C07304=1217.053,344.629,-72.947,-176.067,7.468,148.274
C07305=1217.056,344.381,-72.915,-176.068,7.465,148.273
C07306=1217.060,344.133,-72.884,-176.071,7.462,148.273
C07307=1217.065,343.886,-72.851,-176.073,7.460,148.273
C07308=1217.069,343.638,-72.820,-176.074,7.457,148.273
C07309=1217.073,343.389,-72.787,-176.077,7.454,148.273
C07310=1217.078,343.142,-72.756,-176.078,7.451,148.273
C07311=1217.081,342.894,-72.724,-176.080,7.448,148.272
C07312=1217.086,342.646,-72.691,-176.082,7.445,148.272
C07313=1217.090,342.398,-72.660,-176.084,7.442,148.272
C07314=1217.094,342.150,-72.628,-176.086,7.440,148.272
C07315=1217.098,341.902,-72.596,-176.089,7.436,148.272
C07316=1217.102,341.655,-72.564,-176.090,7.434,148.272
C07317=1217.108,341.376,-72.529,-176.092,7.431,148.271
C07318=1217.112,341.099,-72.493,-176.095,7.427,148.271
C07319=1217.117,340.821,-72.457,-176.097,7.424,148.271
C07320=1217.122,340.543,-72.421,-176.099,7.422,148.271
C07321=1217.126,340.294,-72.390,-176.101,7.418,148.271
C07322=1217.130,340.046,-72.358,-176.103,7.416,148.271
C07323=1217.134,339.799,-72.326,-176.105,7.413,148.271
C07324=1217.138,339.551,-72.294,-176.107,7.410,148.270
C07325=1217.142,339.303,-72.263,-176.109,7.407,148.270
C07326=1217.147,339.055,-72.230,-176.111,7.404,148.270
C07327=1217.151,338.806,-72.199,-176.114,7.401,148.270
C07328=1217.155,338.559,-72.168,-176.115,7.399,148.270
C07329=1217.159,338.311,-72.136,-176.117,7.396,148.270
C07330=1217.164,338.063,-72.104,-176.119,7.393,148.269
C07331=1217.168,337.815,-72.072,-176.121,7.391,148.269
C07332=1217.172,337.567,-72.041,-176.123,7.387,148.269
C07333=1217.176,337.319,-72.010,-176.125,7.385,148.269
C07334=1217.180,337.071,-71.978,-176.128,7.382,148.269
C07335=1217.185,336.824,-71.946,-176.129,7.379,148.269
C07336=1217.189,336.575,-71.914,-176.131,7.376,148.269
C07337=1217.193,336.328,-71.883,-176.134,7.374,148.269
C07338=1217.197,336.080,-71.851,-176.136,7.370,148.268
C07339=1217.201,335.831,-71.820,-176.137,7.368,148.268
C07340=1217.205,335.584,-71.789,-176.140,7.366,148.268
C07341=1217.209,335.336,-71.757,-176.142,7.362,148.268
C07342=1217.214,335.087,-71.725,-176.143,7.360,148.268
C07343=1217.218,334.839,-71.693,-176.146,7.357,148.268
C07344=1217.222,334.591,-71.663,-176.148,7.354,148.268
C07345=1217.226,334.343,-71.631,-176.150,7.351,148.267
C07346=1217.230,334.096,-71.599,-176.152,7.349,148.268
C07347=1217.234,333.847,-71.568,-176.154,7.345,148.267
C07348=1217.239,333.600,-71.537,-176.156,7.343,148.267
C07349=1217.243,333.351,-71.506,-176.158,7.340,148.267
C07350=1217.247,333.104,-71.474,-176.160,7.337,148.267
C07351=1217.252,332.855,-71.442,-176.163,7.334,148.267
C07352=1217.256,332.608,-71.411,-176.164,7.332,148.267
C07353=1217.260,332.360,-71.379,-176.167,7.329,148.267
C07354=1217.264,332.112,-71.348,-176.169,7.326,148.267
C07355=1217.268,331.864,-71.317,-176.171,7.324,148.267
C07356=1217.273,331.616,-71.286,-176.173,7.320,148.266
C07357=1217.277,331.367,-71.255,-176.175,7.318,148.266
C07358=1217.281,331.120,-71.223,-176.177,7.315,148.266
C07359=1217.286,330.872,-71.192,-176.179,7.312,148.266
C07360=1217.289,330.624,-71.161,-176.182,7.309,148.266
C07361=1217.294,330.376,-71.130,-176.183,7.307,148.266
C07362=1217.298,330.128,-71.098,-176.186,7.304,148.266
C07363=1217.302,329.880,-71.067,-176.188,7.301,148.266
C07364=1217.306,329.631,-71.036,-176.190,7.298,148.266
C07365=1217.311,329.384,-71.005,-176.192,7.296,148.266
C07366=1217.315,329.136,-70.974,-176.195,7.293,148.266
C07367=1217.319,328.888,-70.942,-176.196,7.290,148.265
C07368=1217.323,328.640,-70.911,-176.198,7.288,148.265
C07369=1217.328,328.391,-70.880,-176.201,7.284,148.265
C07370=1217.332,328.144,-70.849,-176.203,7.282,148.265
C07371=1217.336,327.895,-70.817,-176.205,7.279,148.265
C07372=1217.340,327.647,-70.787,-176.207,7.277,148.265
C07373=1217.344,327.400,-70.756,-176.210,7.274,148.265
C07374=1217.348,327.151,-70.725,-176.211,7.271,148.265
C07375=1217.353,326.904,-70.694,-176.214,7.268,148.265
C07376=1217.357,326.656,-70.663,-176.216,7.266,148.265
C07377=1217.361,326.407,-70.632,-176.218,7.262,148.265
C07378=1217.366,326.160,-70.601,-176.220,7.260,148.265
C07379=1217.370,325.911,-70.569,-176.222,7.257,148.264
C07380=1217.373,325.663,-70.539,-176.225,7.255,148.265
C07381=1217.378,325.415,-70.508,-176.227,7.251,148.264
C07382=1217.382,325.167,-70.477,-176.229,7.249,148.264
C07383=1217.386,324.919,-70.446,-176.232,7.246,148.264
C07384=1217.391,324.671,-70.415,-176.233,7.244,148.264
C07385=1217.395,324.423,-70.384,-176.235,7.241,148.264
C07386=1217.399,324.175,-70.354,-176.238,7.238,148.264
C07387=1217.403,323.927,-70.323,-176.240,7.236,148.264
C07388=1217.408,323.678,-70.292,-176.242,7.233,148.264
C07389=1217.412,323.430,-70.261,-176.244,7.230,148.264
C07390=1217.416,323.183,-70.230,-176.247,7.227,148.264
C07391=1217.420,322.935,-70.199,-176.249,7.225,148.264
C07392=1217.424,322.687,-70.168,-176.251,7.222,148.264
C07393=1217.429,322.439,-70.138,-176.253,7.219,148.264
C07394=1217.433,322.190,-70.106,-176.256,7.216,148.264
C07395=1217.437,321.943,-70.076,-176.257,7.214,148.264
C07396=1217.441,321.695,-70.046,-176.260,7.211,148.264
C07397=1217.445,321.446,-70.014,-176.262,7.209,148.264
C07398=1217.450,321.198,-69.984,-176.264,7.205,148.263
C07399=1217.454,320.950,-69.953,-176.266,7.203,148.263
C07400=1217.459,320.702,-69.923,-176.269,7.200,148.263
C07401=1217.463,320.454,-69.892,-176.271,7.198,148.264
C07402=1217.466,320.206,-69.861,-176.273,7.195,148.263
C07403=1217.471,319.958,-69.831,-176.275,7.192,148.263
C07404=1217.476,319.710,-69.800,-176.278,7.190,148.263
C07405=1217.479,319.461,-69.770,-176.280,7.187,148.263
C07406=1217.484,319.213,-69.739,-176.282,7.184,148.263
C07407=1217.488,318.965,-69.709,-176.285,7.181,148.263
C07408=1217.492,318.718,-69.678,-176.287,7.179,148.263
C07409=1217.496,318.469,-69.647,-176.289,7.176,148.263
C07410=1217.501,318.221,-69.616,-176.291,7.174,148.263
C07411=1217.505,317.973,-69.586,-176.294,7.171,148.263
C07412=1217.509,317.725,-69.556,-176.296,7.168,148.263
C07413=1217.513,317.476,-69.526,-176.298,7.165,148.263
C07414=1217.518,317.228,-69.495,-176.300,7.163,148.263
C07415=1217.522,316.980,-69.464,-176.302,7.161,148.263
C07416=1217.526,316.733,-69.434,-176.305,7.157,148.263
C07417=1217.531,316.485,-69.403,-176.307,7.155,148.263
C07418=1217.534,316.236,-69.373,-176.309,7.152,148.263
C07419=1217.539,315.988,-69.343,-176.311,7.150,148.263
C07420=1217.544,315.740,-69.312,-176.314,7.147,148.263
C07421=1217.548,315.464,-69.279,-176.317,7.144,148.263
C07422=1217.553,315.188,-69.245,-176.319,7.141,148.263
C07423=1217.558,314.912,-69.211,-176.321,7.138,148.263
C07424=1217.562,314.636,-69.177,-176.324,7.135,148.263
C07425=1217.566,314.388,-69.147,-176.327,7.132,148.263
C07426=1217.571,314.140,-69.117,-176.328,7.130,148.263
C07427=1217.575,313.892,-69.086,-176.331,7.127,148.263
C07428=1217.579,313.644,-69.056,-176.333,7.124,148.263
C07429=1217.584,313.396,-69.026,-176.335,7.122,148.263
C07430=1217.587,313.147,-68.996,-176.338,7.119,148.263
C07431=1217.592,312.899,-68.966,-176.340,7.117,148.263
C07432=1217.596,312.651,-68.935,-176.343,7.114,148.263
C07433=1217.601,312.403,-68.905,-176.344,7.111,148.263
C07434=1217.605,312.155,-68.875,-176.347,7.108,148.263
C07435=1217.609,311.907,-68.844,-176.349,7.106,148.263
C07436=1217.614,311.659,-68.815,-176.352,7.103,148.263
C07437=1217.618,311.411,-68.784,-176.354,7.101,148.263
C07438=1217.622,311.163,-68.755,-176.357,7.098,148.263
C07439=1217.626,310.914,-68.724,-176.359,7.096,148.263
C07440=1217.631,310.666,-68.694,-176.361,7.093,148.263
C07441=1217.635,310.418,-68.664,-176.363,7.090,148.263
C07442=1217.639,310.169,-68.634,-176.366,7.088,148.263
C07443=1217.643,309.922,-68.604,-176.368,7.085,148.263
C07444=1217.648,309.674,-68.574,-176.370,7.083,148.263
C07445=1217.652,309.426,-68.544,-176.373,7.080,148.263
C07446=1217.656,309.177,-68.514,-176.375,7.077,148.263
C07447=1217.660,308.929,-68.485,-176.377,7.074,148.263
C07448=1217.665,308.681,-68.454,-176.379,7.072,148.263
C07449=1217.669,308.433,-68.424,-176.382,7.070,148.263
C07450=1217.673,308.185,-68.394,-176.384,7.067,148.263
C07451=1217.678,307.937,-68.364,-176.386,7.065,148.263
C07452=1217.682,307.688,-68.335,-176.389,7.062,148.263
C07453=1217.686,307.441,-68.305,-176.391,7.059,148.263
C07454=1217.691,307.192,-68.275,-176.394,7.056,148.263
C07455=1217.695,306.944,-68.245,-176.396,7.054,148.263
C07456=1217.699,306.696,-68.215,-176.399,7.051,148.263
C07457=1217.704,306.448,-68.185,-176.401,7.049,148.263
C07458=1217.708,306.199,-68.155,-176.403,7.047,148.263
C07459=1217.712,305.951,-68.126,-176.406,7.044,148.263
C07460=1217.716,305.703,-68.096,-176.408,7.041,148.263
C07461=1217.721,305.455,-68.066,-176.410,7.038,148.263
C07462=1217.725,305.207,-68.036,-176.412,7.036,148.264
C07463=1217.730,304.958,-68.007,-176.415,7.033,148.264
C07464=1217.733,304.711,-67.977,-176.417,7.031,148.264
C07465=1217.738,304.462,-67.947,-176.419,7.029,148.264
C07466=1217.743,304.214,-67.917,-176.422,7.026,148.264
C07467=1217.747,303.966,-67.888,-176.424,7.023,148.264
C07468=1217.751,303.717,-67.858,-176.427,7.020,148.264
C07469=1217.755,303.470,-67.828,-176.429,7.018,148.264
C07470=1217.760,303.221,-67.798,-176.432,7.015,148.264
C07471=1217.764,302.973,-67.769,-176.434,7.013,148.264
C07472=1217.768,302.725,-67.739,-176.436,7.011,148.264
C07473=1217.772,302.476,-67.710,-176.438,7.008,148.264
C07474=1217.776,302.228,-67.680,-176.441,7.006,148.264
C07475=1217.781,301.980,-67.651,-176.443,7.002,148.264
C07476=1217.785,301.731,-67.621,-176.445,7.000,148.264
C07477=1217.790,301.483,-67.591,-176.448,6.997,148.264
C07478=1217.794,301.235,-67.562,-176.451,6.995,148.264
C07479=1217.799,300.987,-67.533,-176.453,6.993,148.264
C07480=1217.803,300.739,-67.503,-176.455,6.990,148.264
C07481=1217.807,300.490,-67.474,-176.458,6.988,148.264
C07482=1217.811,300.242,-67.444,-176.460,6.985,148.264
C07483=1217.815,299.994,-67.415,-176.462,6.983,148.265
C07484=1217.820,299.746,-67.386,-176.464,6.980,148.265
C07485=1217.824,299.497,-67.356,-176.467,6.977,148.265
C07486=1217.828,299.249,-67.327,-176.469,6.975,148.265
C07487=1217.832,299.001,-67.297,-176.472,6.972,148.265
C07488=1217.837,298.753,-67.268,-176.474,6.970,148.265
C07489=1217.842,298.505,-67.238,-176.477,6.968,148.265
C07490=1217.846,298.256,-67.209,-176.479,6.965,148.265
C07491=1217.850,298.008,-67.179,-176.481,6.963,148.265
C07492=1217.854,297.760,-67.150,-176.484,6.960,148.265
C07493=1217.859,297.512,-67.120,-176.486,6.958,148.265
C07494=1217.863,297.263,-67.091,-176.488,6.955,148.265
C07495=1217.868,297.015,-67.062,-176.491,6.952,148.265
C07496=1217.871,296.767,-67.034,-176.494,6.950,148.266
C07497=1217.875,296.519,-67.004,-176.496,6.947,148.266
C07498=1217.880,296.271,-66.975,-176.498,6.945,148.266
C07499=1217.884,296.022,-66.945,-176.500,6.943,148.266
C07500=1217.888,295.774,-66.916,-176.503,6.940,148.266
C07501=1217.893,295.526,-66.887,-176.505,6.938,148.266
C07502=1217.897,295.278,-66.858,-176.508,6.935,148.266
C07503=1217.901,295.029,-66.828,-176.511,6.933,148.266
C07504=1217.906,294.781,-66.799,-176.513,6.931,148.266
C07505=1217.910,294.532,-66.770,-176.515,6.927,148.266
C07506=1217.915,294.285,-66.741,-176.517,6.925,148.266
C07507=1217.919,294.036,-66.712,-176.520,6.922,148.266
C07508=1217.924,293.788,-66.683,-176.523,6.920,148.266
C07509=1217.927,293.540,-66.654,-176.525,6.918,148.267
C07510=1217.931,293.291,-66.625,-176.528,6.915,148.267
C07511=1217.936,293.043,-66.596,-176.530,6.913,148.267
C07512=1217.940,292.795,-66.567,-176.532,6.911,148.267
C07513=1217.945,292.547,-66.537,-176.535,6.908,148.267
C07514=1217.949,292.298,-66.509,-176.537,6.906,148.267
C07515=1217.954,292.050,-66.480,-176.540,6.903,148.267
C07516=1217.957,291.802,-66.451,-176.542,6.901,148.267
C07517=1217.962,291.553,-66.422,-176.544,6.899,148.267
C07518=1217.966,291.305,-66.393,-176.547,6.896,148.267
C07519=1217.971,291.057,-66.364,-176.549,6.893,148.267
C07520=1217.975,290.809,-66.335,-176.551,6.891,148.267
C07521=1217.979,290.560,-66.307,-176.554,6.888,148.267
C07522=1217.984,290.312,-66.277,-176.557,6.886,148.268
C07523=1217.988,290.064,-66.248,-176.559,6.883,148.268
C07524=1217.992,289.815,-66.219,-176.561,6.881,148.268
C07525=1217.997,289.541,-66.188,-176.565,6.878,148.268
C07526=1218.002,289.267,-66.155,-176.567,6.876,148.268
C07527=1218.007,288.993,-66.124,-176.569,6.873,148.268
C07528=1218.011,288.719,-66.092,-176.572,6.870,148.268
C07529=1218.016,288.470,-66.064,-176.575,6.868,148.268
C07530=1218.020,288.222,-66.035,-176.577,6.866,148.269
C07531=1218.024,287.973,-66.006,-176.580,6.863,148.269
C07532=1218.029,287.726,-65.977,-176.582,6.861,148.269
C07533=1218.033,287.477,-65.949,-176.585,6.858,148.269
C07534=1218.037,287.229,-65.919,-176.587,6.856,148.269
C07535=1218.042,286.981,-65.891,-176.589,6.854,148.269
C07536=1218.046,286.732,-65.863,-176.592,6.851,148.269
C07537=1218.050,286.484,-65.833,-176.594,6.849,148.269
C07538=1218.055,286.236,-65.805,-176.597,6.847,148.270
C07539=1218.059,285.987,-65.777,-176.599,6.844,148.270
C07540=1218.064,285.740,-65.748,-176.602,6.841,148.270
C07541=1218.068,285.491,-65.719,-176.604,6.839,148.270
C07542=1218.072,285.242,-65.691,-176.607,6.837,148.270
C07543=1218.077,284.994,-65.663,-176.609,6.834,148.270
C07544=1218.081,284.746,-65.633,-176.611,6.832,148.270
C07545=1218.085,284.497,-65.605,-176.614,6.829,148.270
C07546=1218.090,284.249,-65.577,-176.616,6.827,148.270
C07547=1218.094,284.000,-65.548,-176.618,6.825,148.270
C07548=1218.099,283.753,-65.519,-176.622,6.822,148.271
C07549=1218.103,283.504,-65.491,-176.624,6.820,148.271
C07550=1218.107,283.256,-65.463,-176.626,6.818,148.271
C07551=1218.112,283.007,-65.434,-176.629,6.815,148.271
C07552=1218.116,282.759,-65.406,-176.631,6.813,148.271
C07553=1218.121,282.511,-65.377,-176.633,6.811,148.271
C07554=1218.124,282.263,-65.349,-176.636,6.808,148.271
C07555=1218.129,282.014,-65.320,-176.639,6.806,148.272
C07556=1218.133,281.766,-65.292,-176.641,6.804,148.272
C07557=1218.138,281.518,-65.264,-176.644,6.801,148.272
C07558=1218.142,281.269,-65.236,-176.646,6.799,148.272
C07559=1218.146,281.020,-65.207,-176.648,6.796,148.272
C07560=1218.151,280.772,-65.179,-176.651,6.794,148.272
C07561=1218.155,280.524,-65.150,-176.653,6.792,148.272
C07562=1218.159,280.276,-65.122,-176.656,6.790,148.273
C07563=1218.164,280.027,-65.093,-176.658,6.787,148.273
C07564=1218.168,279.779,-65.065,-176.661,6.784,148.273
C07565=1218.173,279.530,-65.037,-176.663,6.783,148.273
C07566=1218.177,279.283,-65.009,-176.666,6.780,148.273
C07567=1218.181,279.034,-64.981,-176.668,6.777,148.273
C07568=1218.186,278.786,-64.952,-176.671,6.775,148.273
C07569=1218.190,278.537,-64.924,-176.673,6.773,148.273
C07570=1218.195,278.289,-64.896,-176.676,6.771,148.274
C07571=1218.198,278.040,-64.868,-176.678,6.768,148.274
C07572=1218.203,277.793,-64.840,-176.680,6.766,148.274
C07573=1218.208,277.543,-64.812,-176.683,6.764,148.274
C07574=1218.212,277.295,-64.784,-176.686,6.761,148.274
C07575=1218.216,277.046,-64.755,-176.688,6.759,148.274
C07576=1218.221,276.798,-64.728,-176.690,6.757,148.275
C07577=1218.224,276.550,-64.699,-176.693,6.754,148.275
C07578=1218.230,276.302,-64.671,-176.696,6.752,148.275
C07579=1218.234,276.054,-64.643,-176.698,6.750,148.275
C07580=1218.238,275.805,-64.615,-176.700,6.748,148.275
C07581=1218.243,275.557,-64.587,-176.703,6.745,148.275
C07582=1218.247,275.308,-64.559,-176.706,6.743,148.276
C07583=1218.251,275.060,-64.532,-176.708,6.741,148.276
C07584=1218.256,274.811,-64.503,-176.710,6.738,148.276
C07585=1218.260,274.563,-64.475,-176.713,6.736,148.276
C07586=1218.264,274.315,-64.447,-176.715,6.734,148.276
C07587=1218.268,274.066,-64.420,-176.718,6.732,148.276
C07588=1218.274,273.818,-64.392,-176.720,6.729,148.276
C07589=1218.277,273.569,-64.363,-176.723,6.727,148.277
C07590=1218.282,273.321,-64.336,-176.725,6.725,148.277
C07591=1218.286,273.072,-64.308,-176.728,6.722,148.277
C07592=1218.291,272.824,-64.280,-176.730,6.720,148.277
C07593=1218.295,272.576,-64.252,-176.733,6.718,148.277
C07594=1218.299,272.327,-64.225,-176.735,6.716,148.277
C07595=1218.304,272.079,-64.197,-176.738,6.713,148.277
C07596=1218.309,271.831,-64.168,-176.740,6.711,148.278
C07597=1218.313,271.582,-64.141,-176.743,6.709,148.278
C07598=1218.317,271.334,-64.113,-176.745,6.707,148.278
C07599=1218.321,271.085,-64.085,-176.748,6.704,148.278
C07600=1218.325,270.837,-64.058,-176.750,6.702,148.278
C07601=1218.330,270.589,-64.030,-176.753,6.700,148.279
C07602=1218.335,270.339,-64.002,-176.755,6.698,148.279
C07603=1218.339,270.092,-63.974,-176.758,6.695,148.279
C07604=1218.343,269.844,-63.947,-176.761,6.693,148.279
C07605=1218.347,269.594,-63.919,-176.763,6.691,148.279
C07606=1218.352,269.347,-63.891,-176.765,6.689,148.280
C07607=1218.357,269.098,-63.864,-176.768,6.686,148.280
C07608=1218.361,268.849,-63.836,-176.771,6.684,148.280
C07609=1218.365,268.601,-63.809,-176.773,6.682,148.280
C07610=1218.370,268.353,-63.781,-176.775,6.680,148.280
C07611=1218.374,268.104,-63.754,-176.778,6.677,148.280
C07612=1218.378,267.856,-63.726,-176.781,6.675,148.281
C07613=1218.383,267.607,-63.699,-176.783,6.673,148.281
C07614=1218.387,267.359,-63.671,-176.785,6.671,148.281
C07615=1218.391,267.110,-63.643,-176.787,6.669,148.281
C07616=1218.396,266.862,-63.616,-176.791,6.666,148.281
C07617=1218.401,266.614,-63.588,-176.793,6.664,148.281
C07618=1218.406,266.365,-63.561,-176.795,6.662,148.282
C07619=1218.409,266.116,-63.533,-176.797,6.660,148.282
C07620=1218.414,265.868,-63.506,-176.801,6.657,148.282
C07621=1218.418,265.620,-63.478,-176.803,6.655,148.282
C07622=1218.423,265.372,-63.451,-176.805,6.653,148.282
C07623=1218.427,265.122,-63.423,-176.807,6.651,148.282
C07624=1218.431,264.875,-63.396,-176.810,6.649,148.283
C07625=1218.436,264.626,-63.369,-176.813,6.646,148.283
C07626=1218.441,264.378,-63.342,-176.815,6.644,148.283
C07627=1218.445,264.129,-63.313,-176.818,6.642,148.283
C07628=1218.449,263.880,-63.286,-176.820,6.640,148.283
C07629=1218.454,263.608,-63.257,-176.823,6.637,148.284
C07630=1218.459,263.336,-63.226,-176.826,6.635,148.284
C07631=1218.464,263.063,-63.197,-176.829,6.632,148.284
C07632=1218.469,262.789,-63.167,-176.831,6.630,148.284
C07633=1218.473,262.541,-63.140,-176.834,6.628,148.285
C07634=1218.477,262.293,-63.112,-176.836,6.625,148.285
C07635=1218.481,262.045,-63.085,-176.839,6.624,148.285
C07636=1218.486,261.796,-63.058,-176.841,6.621,148.285
C07637=1218.490,261.547,-63.031,-176.844,6.620,148.285
C07638=1218.495,261.299,-63.004,-176.846,6.617,148.285
C07639=1218.499,261.051,-62.976,-176.849,6.615,148.286
C07640=1218.504,260.802,-62.949,-176.852,6.613,148.286
C07641=1218.508,260.554,-62.922,-176.854,6.611,148.286
C07642=1218.513,260.305,-62.895,-176.856,6.609,148.286
C07643=1218.516,260.056,-62.868,-176.859,6.606,148.286
C07644=1218.521,259.808,-62.841,-176.862,6.604,148.287
C07645=1218.526,259.559,-62.814,-176.864,6.602,148.287
C07646=1218.530,259.311,-62.787,-176.867,6.600,148.287
C07647=1218.535,259.063,-62.759,-176.869,6.598,148.287
C07648=1218.539,258.814,-62.732,-176.871,6.596,148.288
C07649=1218.543,258.566,-62.705,-176.874,6.594,148.288
C07650=1218.547,258.317,-62.678,-176.877,6.591,148.288
C07651=1218.552,258.069,-62.651,-176.879,6.589,148.288
C07652=1218.557,257.820,-62.624,-176.882,6.587,148.288
C07653=1218.561,257.572,-62.597,-176.884,6.585,148.289
C07654=1218.565,257.323,-62.570,-176.887,6.583,148.289
C07655=1218.570,257.075,-62.543,-176.889,6.581,148.289
C07656=1218.575,256.826,-62.516,-176.892,6.578,148.289
C07657=1218.579,256.578,-62.489,-176.894,6.576,148.289
C07658=1218.583,256.330,-62.463,-176.897,6.574,148.290
C07659=1218.588,256.081,-62.436,-176.899,6.572,148.290
C07660=1218.592,255.832,-62.408,-176.902,6.570,148.290
C07661=1218.597,255.583,-62.382,-176.904,6.568,148.290
C07662=1218.601,255.335,-62.355,-176.907,6.565,148.291
C07663=1218.605,255.086,-62.328,-176.910,6.563,148.291
C07664=1218.610,254.838,-62.301,-176.912,6.561,148.291
C07665=1218.614,254.590,-62.275,-176.914,6.559,148.291
C07666=1218.619,254.341,-62.248,-176.917,6.557,148.291
C07667=1218.623,254.093,-62.221,-176.919,6.555,148.292
C07668=1218.627,253.844,-62.194,-176.922,6.553,148.292
C07669=1218.632,253.595,-62.168,-176.925,6.550,148.292
C07670=1218.637,253.347,-62.141,-176.927,6.548,148.292
C07671=1218.641,253.099,-62.114,-176.930,6.547,148.293
C07672=1218.645,252.850,-62.087,-176.932,6.544,148.293
C07673=1218.650,252.602,-62.060,-176.935,6.543,148.293
C07674=1218.654,252.353,-62.035,-176.937,6.541,148.293
C07675=1218.659,252.104,-62.007,-176.939,6.538,148.293
C07676=1218.664,251.856,-61.980,-176.942,6.536,148.294
C07677=1218.668,251.608,-61.954,-176.945,6.534,148.294
C07678=1218.672,251.358,-61.928,-176.947,6.532,148.294
C07679=1218.676,251.110,-61.901,-176.950,6.530,148.294
C07680=1218.681,250.862,-61.874,-176.952,6.528,148.295
C07681=1218.685,250.613,-61.848,-176.955,6.526,148.295
C07682=1218.690,250.365,-61.821,-176.957,6.524,148.295
C07683=1218.695,250.116,-61.794,-176.960,6.522,148.295
C07684=1218.699,249.867,-61.768,-176.962,6.519,148.295
C07685=1218.703,249.619,-61.741,-176.965,6.517,148.296
C07686=1218.707,249.371,-61.715,-176.968,6.515,148.296
C07687=1218.712,249.121,-61.689,-176.970,6.513,148.296
C07688=1218.716,248.873,-61.662,-176.972,6.511,148.296
C07689=1218.721,248.624,-61.636,-176.975,6.509,148.297
C07690=1218.725,248.376,-61.609,-176.977,6.507,148.297
C07691=1218.730,248.127,-61.582,-176.980,6.505,148.297
C07692=1218.734,247.879,-61.556,-176.982,6.503,148.297
C07693=1218.739,247.630,-61.529,-176.985,6.500,148.298
C07694=1218.743,247.381,-61.504,-176.988,6.499,148.298
C07695=1218.748,247.134,-61.477,-176.990,6.497,148.298
C07696=1218.752,246.885,-61.451,-176.993,6.495,148.298
C07697=1218.757,246.636,-61.424,-176.995,6.493,148.299
C07698=1218.761,246.387,-61.398,-176.998,6.491,148.299
C07699=1218.766,246.139,-61.371,-177.000,6.489,148.299
C07700=1218.770,245.890,-61.346,-177.002,6.487,148.299
C07701=1218.774,245.642,-61.319,-177.005,6.485,148.300
C07702=1218.779,245.393,-61.293,-177.008,6.483,148.300
C07703=1218.783,245.145,-61.266,-177.010,6.481,148.300
C07704=1218.788,244.896,-61.240,-177.013,6.478,148.300
C07705=1218.792,244.648,-61.214,-177.016,6.476,148.301
C07706=1218.797,244.399,-61.188,-177.018,6.474,148.301
C07707=1218.802,244.150,-61.162,-177.020,6.472,148.301
C07708=1218.806,243.902,-61.135,-177.023,6.470,148.301
C07709=1218.810,243.653,-61.110,-177.026,6.468,148.302
C07710=1218.815,243.404,-61.083,-177.028,6.467,148.302
C07711=1218.819,243.156,-61.057,-177.030,6.464,148.302
C07712=1218.824,242.907,-61.031,-177.033,6.462,148.302
C07713=1218.828,242.659,-61.005,-177.036,6.461,148.303
C07714=1218.832,242.410,-60.979,-177.038,6.459,148.303
C07715=1218.837,242.161,-60.952,-177.040,6.457,148.303
C07716=1218.842,241.913,-60.926,-177.043,6.455,148.303
C07717=1218.845,241.664,-60.900,-177.046,6.452,148.304
C07718=1218.850,241.416,-60.875,-177.049,6.450,148.304
C07719=1218.855,241.167,-60.848,-177.051,6.448,148.304
C07720=1218.860,240.918,-60.822,-177.054,6.446,148.304
C07721=1218.863,240.670,-60.796,-177.056,6.444,148.305
C07722=1218.868,240.421,-60.770,-177.059,6.442,148.305
C07723=1218.873,240.173,-60.744,-177.061,6.440,148.305
C07724=1218.877,239.924,-60.719,-177.064,6.438,148.305
C07725=1218.881,239.676,-60.692,-177.066,6.436,148.306
C07726=1218.886,239.427,-60.666,-177.069,6.435,148.306
C07727=1218.891,239.178,-60.640,-177.071,6.432,148.306
C07728=1218.895,238.930,-60.615,-177.074,6.430,148.306
C07729=1218.900,238.681,-60.589,-177.076,6.429,148.307
C07730=1218.904,238.432,-60.563,-177.079,6.427,148.307
C07731=1218.908,238.184,-60.536,-177.081,6.425,148.307
C07732=1218.913,237.936,-60.511,-177.084,6.423,148.307
C07733=1218.918,237.664,-60.483,-177.087,6.420,148.308
C07734=1218.923,237.392,-60.455,-177.089,6.418,148.308
C07735=1218.928,237.121,-60.426,-177.092,6.416,148.308
C07736=1218.932,236.849,-60.398,-177.095,6.414,148.309
C07737=1218.937,236.601,-60.373,-177.098,6.412,148.309
C07738=1218.942,236.352,-60.346,-177.100,6.410,148.309
C07739=1218.946,236.103,-60.321,-177.103,6.408,148.309
C07740=1218.951,235.855,-60.295,-177.105,6.406,148.310
C07741=1218.955,235.606,-60.270,-177.108,6.404,148.310
C07742=1218.960,235.358,-60.244,-177.110,6.402,148.310
C07743=1218.964,235.109,-60.218,-177.113,6.400,148.311
C07744=1218.969,234.861,-60.193,-177.115,6.398,148.311
C07745=1218.973,234.612,-60.167,-177.118,6.396,148.311
C07746=1218.977,234.363,-60.141,-177.120,6.394,148.311
C07747=1218.983,234.115,-60.115,-177.123,6.392,148.312
C07748=1218.987,233.866,-60.089,-177.126,6.391,148.312
C07749=1218.991,233.617,-60.064,-177.128,6.388,148.312
C07750=1218.995,233.368,-60.038,-177.130,6.387,148.312
C07751=1219.000,233.120,-60.012,-177.133,6.385,148.313
C07752=1219.004,232.871,-59.987,-177.136,6.383,148.313
C07753=1219.009,232.623,-59.961,-177.138,6.381,148.313
C07754=1219.014,232.374,-59.936,-177.141,6.379,148.314
C07755=1219.018,232.125,-59.911,-177.143,6.377,148.314
C07756=1219.023,231.877,-59.885,-177.146,6.375,148.314
C07757=1219.027,231.628,-59.859,-177.148,6.373,148.314
C07758=1219.031,231.379,-59.834,-177.151,6.371,148.315
C07759=1219.036,231.131,-59.808,-177.154,6.369,148.315
C07760=1219.041,230.882,-59.783,-177.156,6.367,148.315
C07761=1219.045,230.633,-59.758,-177.158,6.365,148.316
C07762=1219.050,230.385,-59.732,-177.161,6.364,148.316
C07763=1219.054,230.136,-59.706,-177.164,6.362,148.316
C07764=1219.059,229.888,-59.681,-177.166,6.360,148.317
C07765=1219.063,229.639,-59.656,-177.169,6.358,148.317
C07766=1219.068,229.390,-59.630,-177.171,6.356,148.317
C07767=1219.072,229.142,-59.605,-177.174,6.354,148.317
C07768=1219.077,228.892,-59.580,-177.176,6.352,148.318
C07769=1219.082,228.644,-59.554,-177.179,6.350,148.318
C07770=1219.085,228.396,-59.529,-177.182,6.348,148.318
C07771=1219.089,228.147,-59.503,-177.184,6.347,148.319
C07772=1219.095,227.898,-59.479,-177.187,6.345,148.319
C07773=1219.099,227.649,-59.453,-177.189,6.342,148.319
C07774=1219.104,227.401,-59.428,-177.192,6.341,148.319
C07775=1219.108,227.152,-59.403,-177.194,6.339,148.320
C07776=1219.113,226.904,-59.377,-177.197,6.337,148.320
C07777=1219.117,226.654,-59.352,-177.199,6.335,148.320
C07778=1219.122,226.406,-59.327,-177.202,6.333,148.321
C07779=1219.126,226.158,-59.302,-177.205,6.331,148.321
C07780=1219.130,225.908,-59.277,-177.207,6.329,148.321
C07781=1219.135,225.660,-59.251,-177.209,6.327,148.321
C07782=1219.140,225.411,-59.226,-177.212,6.325,148.322
C07783=1219.145,225.163,-59.201,-177.215,6.324,148.322
C07784=1219.148,224.914,-59.176,-177.217,6.322,148.322
C07785=1219.153,224.665,-59.151,-177.220,6.320,148.323
C07786=1219.158,224.416,-59.126,-177.223,6.318,148.323
C07787=1219.162,224.168,-59.101,-177.225,6.316,148.323
C07788=1219.167,223.918,-59.076,-177.228,6.314,148.324
C07789=1219.171,223.671,-59.051,-177.231,6.312,148.324
C07790=1219.176,223.421,-59.026,-177.233,6.310,148.324
C07791=1219.180,223.173,-59.000,-177.235,6.308,148.324
C07792=1219.185,222.924,-58.975,-177.238,6.307,148.325
C07793=1219.189,222.676,-58.951,-177.241,6.305,148.325
C07794=1219.194,222.426,-58.926,-177.243,6.303,148.325
C07795=1219.198,222.178,-58.900,-177.246,6.301,148.326
C07796=1219.203,221.929,-58.875,-177.248,6.299,148.326
C07797=1219.207,221.681,-58.851,-177.251,6.297,148.326
C07798=1219.212,221.432,-58.826,-177.254,6.295,148.327
C07799=1219.217,221.183,-58.801,-177.256,6.294,148.327
C07800=1219.221,220.935,-58.776,-177.258,6.291,148.327
C07801=1219.225,220.686,-58.751,-177.261,6.290,148.327
C07802=1219.230,220.437,-58.726,-177.263,6.289,148.328
C07803=1219.234,220.189,-58.701,-177.266,6.287,148.328
C07804=1219.239,219.940,-58.676,-177.268,6.285,148.328
C07805=1219.244,219.690,-58.651,-177.271,6.283,148.329
C07806=1219.248,219.443,-58.626,-177.274,6.281,148.329
C07807=1219.253,219.194,-58.602,-177.276,6.279,148.329
C07808=1219.257,218.944,-58.577,-177.279,6.277,148.330
C07809=1219.262,218.696,-58.553,-177.282,6.276,148.330
C07810=1219.266,218.447,-58.527,-177.284,6.274,148.330
C07811=1219.271,218.199,-58.502,-177.287,6.272,148.331
C07812=1219.276,217.950,-58.478,-177.290,6.270,148.331
C07813=1219.280,217.701,-58.453,-177.292,6.268,148.331
C07814=1219.284,217.453,-58.428,-177.295,6.266,148.332
C07815=1219.289,217.203,-58.403,-177.297,6.264,148.332
C07816=1219.294,216.955,-58.379,-177.300,6.262,148.332
C07817=1219.298,216.706,-58.355,-177.302,6.260,148.333
C07818=1219.303,216.457,-58.330,-177.305,6.259,148.333
C07819=1219.307,216.209,-58.305,-177.307,6.257,148.333
C07820=1219.312,215.960,-58.280,-177.310,6.255,148.334
C07821=1219.316,215.711,-58.256,-177.313,6.253,148.334
C07822=1219.321,215.463,-58.231,-177.315,6.252,148.334
C07823=1219.325,215.214,-58.207,-177.317,6.250,148.335
C07824=1219.330,214.965,-58.182,-177.320,6.248,148.335
C07825=1219.334,214.716,-58.158,-177.323,6.246,148.335
C07826=1219.339,214.468,-58.133,-177.325,6.245,148.336
C07827=1219.343,214.218,-58.109,-177.328,6.243,148.336
C07828=1219.348,213.970,-58.084,-177.331,6.241,148.336
C07829=1219.353,213.721,-58.060,-177.333,6.239,148.337
C07830=1219.357,213.472,-58.035,-177.336,6.237,148.337
C07831=1219.361,213.224,-58.010,-177.339,6.235,148.337
C07832=1219.366,212.975,-57.985,-177.341,6.233,148.338
C07833=1219.370,212.726,-57.961,-177.344,6.232,148.338
C07834=1219.375,212.478,-57.936,-177.346,6.230,148.338
C07835=1219.380,212.229,-57.912,-177.349,6.228,148.339
C07836=1219.385,211.980,-57.888,-177.351,6.227,148.339
C07837=1219.389,211.709,-57.862,-177.354,6.224,148.339
C07838=1219.394,211.439,-57.835,-177.357,6.222,148.340
C07839=1219.399,211.169,-57.808,-177.360,6.221,148.340
C07840=1219.404,210.899,-57.782,-177.362,6.219,148.340
C07841=1219.409,210.649,-57.758,-177.365,6.217,148.341
C07842=1219.414,210.400,-57.733,-177.368,6.215,148.341
C07843=1219.418,210.152,-57.709,-177.370,6.213,148.341
C07844=1219.422,209.903,-57.685,-177.373,6.211,148.342
C07845=1219.427,209.654,-57.660,-177.375,6.209,148.342
C07846=1219.431,209.406,-57.636,-177.378,6.208,148.342
C07847=1219.436,209.157,-57.612,-177.380,6.207,148.343
C07848=1219.441,208.909,-57.587,-177.383,6.205,148.343
C07849=1219.445,208.659,-57.564,-177.385,6.203,148.343
C07850=1219.449,208.410,-57.539,-177.388,6.201,148.344
C07851=1219.454,208.162,-57.515,-177.391,6.199,148.344
C07852=1219.459,207.913,-57.491,-177.393,6.197,148.344
C07853=1219.463,207.665,-57.467,-177.396,6.195,148.345
C07854=1219.468,207.415,-57.442,-177.399,6.194,148.345
C07855=1219.473,207.166,-57.418,-177.401,6.192,148.345
C07856=1219.477,206.918,-57.394,-177.403,6.191,148.346
C07857=1219.482,206.669,-57.370,-177.406,6.189,148.346
C07858=1219.487,206.420,-57.346,-177.409,6.187,148.346
C07859=1219.491,206.172,-57.322,-177.412,6.186,148.347
C07860=1219.495,205.923,-57.298,-177.414,6.184,148.347
C07861=1219.500,205.673,-57.274,-177.417,6.182,148.348
C07862=1219.505,205.425,-57.250,-177.420,6.180,148.348
C07863=1219.509,205.176,-57.226,-177.422,6.178,148.348
C07864=1219.514,204.928,-57.201,-177.424,6.177,148.349
C07865=1219.519,204.679,-57.178,-177.427,6.175,148.349
C07866=1219.523,204.430,-57.153,-177.430,6.173,148.349
C07867=1219.527,204.181,-57.130,-177.432,6.172,148.350
C07868=1219.532,203.932,-57.106,-177.435,6.170,148.350
C07869=1219.536,203.684,-57.082,-177.438,6.168,148.350
C07870=1219.542,203.434,-57.058,-177.440,6.166,148.351
C07871=1219.546,203.186,-57.034,-177.442,6.165,148.351
C07872=1219.551,202.937,-57.010,-177.445,6.163,148.351
C07873=1219.555,202.688,-56.986,-177.448,6.161,148.352
C07874=1219.559,202.439,-56.962,-177.450,6.160,148.352
C07875=1219.564,202.190,-56.938,-177.453,6.158,148.352
C07876=1219.569,201.942,-56.914,-177.455,6.156,148.353
C07877=1219.574,201.693,-56.890,-177.458,6.154,148.353
C07878=1219.578,201.444,-56.866,-177.460,6.153,148.353
C07879=1219.583,201.195,-56.843,-177.463,6.151,148.354
C07880=1219.587,200.947,-56.819,-177.466,6.149,148.354
C07881=1219.592,200.698,-56.795,-177.468,6.148,148.354
C07882=1219.596,200.449,-56.771,-177.471,6.146,148.355
C07883=1219.600,200.200,-56.748,-177.473,6.144,148.355
C07884=1219.605,199.951,-56.724,-177.476,6.143,148.356
C07885=1219.609,199.702,-56.700,-177.479,6.141,148.356
C07886=1219.614,199.453,-56.676,-177.481,6.139,148.356
C07887=1219.619,199.204,-56.652,-177.484,6.138,148.357
C07888=1219.624,198.955,-56.629,-177.487,6.136,148.357
C07889=1219.628,198.707,-56.605,-177.489,6.134,148.357
C07890=1219.633,198.458,-56.581,-177.491,6.133,148.358
C07891=1219.637,198.210,-56.557,-177.494,6.131,148.358
C07892=1219.642,197.961,-56.534,-177.497,6.129,148.359
C07893=1219.647,197.711,-56.511,-177.499,6.127,148.359
C07894=1219.651,197.463,-56.486,-177.502,6.126,148.359
C07895=1219.656,197.214,-56.463,-177.505,6.124,148.360
C07896=1219.661,196.965,-56.440,-177.507,6.123,148.360
C07897=1219.665,196.717,-56.416,-177.509,6.121,148.360
C07898=1219.670,196.468,-56.392,-177.512,6.119,148.361
C07899=1219.674,196.219,-56.369,-177.515,6.118,148.361
C07900=1219.679,195.969,-56.346,-177.518,6.116,148.362
C07901=1219.683,195.721,-56.322,-177.520,6.115,148.362
C07902=1219.688,195.472,-56.298,-177.522,6.113,148.362
C07903=1219.693,195.223,-56.275,-177.525,6.111,148.363
C07904=1219.697,194.975,-56.251,-177.528,6.109,148.363
C07905=1219.702,194.726,-56.227,-177.530,6.107,148.363
C07906=1219.707,194.477,-56.204,-177.532,6.106,148.364
C07907=1219.711,194.228,-56.181,-177.535,6.104,148.364
C07908=1219.715,193.979,-56.158,-177.538,6.103,148.364
C07909=1219.720,193.730,-56.134,-177.541,6.101,148.365
C07910=1219.724,193.481,-56.110,-177.543,6.099,148.365
C07911=1219.729,193.232,-56.087,-177.546,6.098,148.366
C07912=1219.734,192.983,-56.064,-177.548,6.096,148.366
C07913=1219.738,192.734,-56.040,-177.551,6.095,148.366
C07914=1219.743,192.485,-56.017,-177.553,6.093,148.367
C07915=1219.748,192.236,-55.994,-177.556,6.091,148.367
C07916=1219.751,191.988,-55.970,-177.558,6.090,148.367
C07917=1219.757,191.740,-55.947,-177.561,6.088,148.368
C07918=1219.761,191.491,-55.924,-177.564,6.086,148.368
C07919=1219.766,191.242,-55.900,-177.567,6.085,148.369
C07920=1219.771,190.993,-55.877,-177.569,6.084,148.369
C07921=1219.776,190.744,-55.854,-177.571,6.082,148.369
C07922=1219.780,190.495,-55.830,-177.574,6.080,148.370
C07923=1219.784,190.246,-55.808,-177.577,6.078,148.370
C07924=1219.789,189.997,-55.784,-177.579,6.076,148.370
C07925=1219.794,189.748,-55.761,-177.581,6.075,148.371
C07926=1219.798,189.499,-55.738,-177.584,6.074,148.371
C07927=1219.804,189.250,-55.715,-177.587,6.072,148.372
C07928=1219.808,189.002,-55.692,-177.590,6.070,148.372
C07929=1219.812,188.753,-55.668,-177.592,6.069,148.372
C07930=1219.817,188.504,-55.645,-177.595,6.067,148.373
C07931=1219.822,188.255,-55.622,-177.597,6.066,148.373
C07932=1219.826,188.006,-55.599,-177.600,6.064,148.374
C07933=1219.830,187.757,-55.576,-177.602,6.063,148.374
C07934=1219.836,187.509,-55.553,-177.605,6.061,148.374
C07935=1219.840,187.259,-55.529,-177.608,6.059,148.375
C07936=1219.844,187.011,-55.507,-177.610,6.058,148.375
C07937=1219.849,186.762,-55.483,-177.612,6.057,148.376
C07938=1219.854,186.512,-55.461,-177.615,6.055,148.376
C07939=1219.858,186.263,-55.438,-177.618,6.053,148.376
C07940=1219.863,186.015,-55.415,-177.620,6.051,148.377
C07941=1219.869,185.745,-55.390,-177.624,6.050,148.377
C07942=1219.873,185.475,-55.365,-177.626,6.048,148.378
C07943=1219.878,185.205,-55.340,-177.629,6.046,148.378
C07944=1219.883,184.936,-55.314,-177.632,6.044,148.378
C07945=1219.888,184.688,-55.292,-177.634,6.043,148.379
C07946=1219.893,184.439,-55.269,-177.637,6.042,148.379
C07947=1219.897,184.189,-55.246,-177.639,6.040,148.380
C07948=1219.901,183.941,-55.223,-177.641,6.039,148.380
C07949=1219.906,183.691,-55.200,-177.644,6.037,148.380
C07950=1219.911,183.443,-55.178,-177.647,6.035,148.381
C07951=1219.915,183.194,-55.155,-177.650,6.034,148.381
C07952=1219.920,182.945,-55.131,-177.652,6.033,148.382
C07953=1219.924,182.696,-55.109,-177.655,6.031,148.382
C07954=1219.930,182.447,-55.086,-177.657,6.029,148.382
C07955=1219.934,182.199,-55.063,-177.660,6.027,148.383
C07956=1219.938,181.950,-55.040,-177.663,6.026,148.383
C07957=1219.943,181.700,-55.018,-177.665,6.025,148.384
C07958=1219.948,181.452,-54.995,-177.668,6.023,148.384
C07959=1219.953,181.203,-54.972,-177.670,6.022,148.384
C07960=1219.957,180.954,-54.950,-177.673,6.020,148.385
C07961=1219.962,180.705,-54.926,-177.676,6.018,148.385
C07962=1219.966,180.457,-54.904,-177.678,6.017,148.386
C07963=1219.971,180.207,-54.881,-177.680,6.016,148.386
C07964=1219.975,179.958,-54.858,-177.683,6.014,148.386
C07965=1219.980,179.708,-54.836,-177.686,6.012,148.387
C07966=1219.985,179.460,-54.813,-177.688,6.011,148.387
C07967=1219.989,179.211,-54.790,-177.691,6.009,148.388
C07968=1219.994,178.962,-54.768,-177.694,6.008,148.388
C07969=1219.999,178.714,-54.745,-177.696,6.007,148.388
C07970=1220.003,178.464,-54.723,-177.698,6.005,148.389
C07971=1220.008,178.215,-54.700,-177.701,6.003,148.389
C07972=1220.013,177.967,-54.678,-177.704,6.002,148.390
C07973=1220.018,177.718,-54.655,-177.706,6.000,148.390
C07974=1220.022,177.468,-54.632,-177.709,5.999,148.390
C07975=1220.027,177.220,-54.609,-177.712,5.997,148.391
C07976=1220.031,176.971,-54.587,-177.714,5.996,148.391
C07977=1220.035,176.722,-54.565,-177.717,5.994,148.392
C07978=1220.041,176.473,-54.542,-177.720,5.992,148.392
C07979=1220.045,176.224,-54.520,-177.722,5.991,148.393
C07980=1220.050,175.975,-54.497,-177.724,5.990,148.393
C07981=1220.054,175.727,-54.475,-177.727,5.988,148.393
C07982=1220.059,175.477,-54.453,-177.729,5.987,148.394
C07983=1220.064,175.228,-54.430,-177.732,5.985,148.394
C07984=1220.068,174.980,-54.408,-177.735,5.984,148.395
C07985=1220.073,174.730,-54.385,-177.737,5.983,148.395
C07986=1220.077,174.481,-54.362,-177.740,5.981,148.396
C07987=1220.082,174.233,-54.340,-177.743,5.979,148.396
C07988=1220.087,173.983,-54.318,-177.745,5.978,148.396
C07989=1220.092,173.735,-54.295,-177.747,5.976,148.397
C07990=1220.096,173.486,-54.273,-177.750,5.975,148.397
C07991=1220.101,173.236,-54.251,-177.753,5.974,148.398
C07992=1220.106,172.988,-54.228,-177.755,5.972,148.398
C07993=1220.110,172.739,-54.206,-177.758,5.970,148.398
C07994=1220.115,172.490,-54.184,-177.760,5.969,148.399
C07995=1220.119,172.241,-54.161,-177.763,5.968,148.399
C07996=1220.124,171.992,-54.139,-177.766,5.966,148.400
C07997=1220.129,171.743,-54.117,-177.768,5.965,148.400
C07998=1220.133,171.494,-54.094,-177.771,5.963,148.400
C07999=1220.138,171.245,-54.072,-177.774,5.962,148.401
C08000=1220.142,170.996,-54.050,-177.776,5.961,148.401
C08001=1220.148,170.747,-54.028,-177.779,5.959,148.402
C08002=1220.152,170.498,-54.006,-177.781,5.958,148.402
C08003=1220.157,170.250,-53.984,-177.784,5.956,148.403
C08004=1220.161,170.000,-53.962,-177.786,5.955,148.403
C08005=1220.166,169.751,-53.939,-177.789,5.954,148.403
C08006=1220.171,169.502,-53.917,-177.791,5.952,148.404
C08007=1220.175,169.253,-53.895,-177.794,5.950,148.404
C08008=1220.180,169.005,-53.873,-177.796,5.949,148.405
C08009=1220.185,168.755,-53.850,-177.799,5.947,148.405
C08010=1220.190,168.506,-53.829,-177.802,5.946,148.406
C08011=1220.194,168.257,-53.806,-177.804,5.945,148.406
C08012=1220.199,168.008,-53.785,-177.807,5.943,148.407
C08013=1220.203,167.759,-53.763,-177.809,5.942,148.407
C08014=1220.209,167.510,-53.740,-177.812,5.940,148.407
C08015=1220.213,167.261,-53.718,-177.815,5.939,148.408
C08016=1220.217,167.013,-53.696,-177.817,5.938,148.408
C08017=1220.222,166.763,-53.674,-177.820,5.936,148.409
C08018=1220.227,166.515,-53.652,-177.822,5.934,148.409
C08019=1220.231,166.265,-53.630,-177.825,5.934,148.410
C08020=1220.236,166.017,-53.609,-177.828,5.932,148.410
C08021=1220.241,165.767,-53.586,-177.830,5.931,148.410
C08022=1220.246,165.518,-53.564,-177.833,5.929,148.411
C08023=1220.250,165.269,-53.542,-177.835,5.927,148.411
C08024=1220.255,165.020,-53.520,-177.838,5.926,148.412
C08025=1220.260,164.772,-53.499,-177.840,5.925,148.412
C08026=1220.264,164.522,-53.477,-177.843,5.924,148.413
C08027=1220.269,164.274,-53.455,-177.845,5.922,148.413
C08028=1220.273,164.024,-53.433,-177.848,5.920,148.413
C08029=1220.278,163.776,-53.411,-177.851,5.920,148.414
C08030=1220.282,163.527,-53.389,-177.853,5.918,148.414
C08031=1220.287,163.278,-53.368,-177.855,5.917,148.415
C08032=1220.292,163.028,-53.345,-177.858,5.915,148.415
C08033=1220.297,162.779,-53.324,-177.861,5.914,148.416
C08034=1220.302,162.530,-53.302,-177.863,5.913,148.416
C08035=1220.306,162.281,-53.280,-177.866,5.911,148.416
C08036=1220.311,162.032,-53.259,-177.869,5.910,148.417
C08037=1220.315,161.783,-53.237,-177.871,5.908,148.417
C08038=1220.320,161.534,-53.215,-177.874,5.906,148.418
C08039=1220.325,161.286,-53.193,-177.876,5.905,148.418
C08040=1220.329,161.036,-53.171,-177.879,5.904,148.419
C08041=1220.335,160.787,-53.150,-177.881,5.903,148.419
C08042=1220.339,160.538,-53.128,-177.884,5.901,148.420
C08043=1220.344,160.289,-53.106,-177.887,5.901,148.420
C08044=1220.349,160.040,-53.085,-177.889,5.899,148.421
C08045=1220.353,159.771,-53.062,-177.892,5.897,148.421
C08046=1220.359,159.503,-53.038,-177.895,5.895,148.422
C08047=1220.363,159.234,-53.015,-177.897,5.894,148.422
C08048=1220.369,158.964,-52.992,-177.900,5.893,148.423
C08049=1220.373,158.715,-52.970,-177.903,5.891,148.423
C08050=1220.378,158.466,-52.948,-177.906,5.890,148.423
C08051=1220.383,158.217,-52.927,-177.908,5.889,148.424
C08052=1220.387,157.968,-52.905,-177.910,5.888,148.424
C08053=1220.392,157.719,-52.883,-177.913,5.886,148.425
C08054=1220.397,157.470,-52.862,-177.916,5.884,148.425
C08055=1220.401,157.221,-52.841,-177.918,5.883,148.426
C08056=1220.406,156.972,-52.819,-177.921,5.882,148.426
C08057=1220.411,156.723,-52.798,-177.924,5.881,148.427
C08058=1220.415,156.474,-52.776,-177.926,5.879,148.427
C08059=1220.420,156.225,-52.755,-177.929,5.878,148.428
C08060=1220.425,155.976,-52.734,-177.931,5.877,148.428
C08061=1220.430,155.726,-52.712,-177.934,5.876,148.428
C08062=1220.434,155.478,-52.690,-177.937,5.874,148.429
C08063=1220.439,155.229,-52.669,-177.939,5.872,148.429
C08064=1220.443,154.979,-52.647,-177.941,5.871,148.430
C08065=1220.448,154.731,-52.626,-177.945,5.870,148.430
C08066=1220.453,154.481,-52.605,-177.947,5.869,148.431
C08067=1220.458,154.233,-52.583,-177.949,5.867,148.431
C08068=1220.462,153.983,-52.562,-177.952,5.866,148.432
C08069=1220.467,153.735,-52.541,-177.955,5.865,148.432
C08070=1220.472,153.485,-52.520,-177.957,5.864,148.432
C08071=1220.477,153.237,-52.498,-177.960,5.862,148.433
C08072=1220.481,152.987,-52.477,-177.962,5.861,148.433
C08073=1220.486,152.738,-52.456,-177.965,5.859,148.434
C08074=1220.491,152.489,-52.435,-177.967,5.859,148.434
C08075=1220.496,152.240,-52.413,-177.970,5.857,148.435
C08076=1220.500,151.990,-52.392,-177.973,5.855,148.435
C08077=1220.504,151.742,-52.371,-177.975,5.854,148.436
C08078=1220.509,151.493,-52.350,-177.978,5.853,148.436
C08079=1220.514,151.244,-52.328,-177.980,5.852,148.437
C08080=1220.520,150.995,-52.307,-177.983,5.850,148.437
C08081=1220.523,150.746,-52.285,-177.985,5.849,148.438
C08082=1220.528,150.497,-52.265,-177.988,5.848,148.438
C08083=1220.533,150.247,-52.244,-177.990,5.847,148.439
C08084=1220.538,149.999,-52.222,-177.993,5.845,148.439
C08085=1220.542,149.749,-52.201,-177.996,5.844,148.440
C08086=1220.547,149.501,-52.179,-177.998,5.843,148.440
C08087=1220.552,149.251,-52.158,-178.001,5.842,148.440
C08088=1220.557,149.002,-52.138,-178.004,5.840,148.441
C08089=1220.561,148.754,-52.116,-178.006,5.839,148.441
C08090=1220.567,148.504,-52.095,-178.009,5.838,148.442
C08091=1220.570,148.255,-52.075,-178.011,5.837,148.442
C08092=1220.575,148.006,-52.053,-178.014,5.835,148.443
C08093=1220.581,147.757,-52.032,-178.016,5.834,148.443
C08094=1220.585,147.508,-52.012,-178.019,5.832,148.444
C08095=1220.590,147.259,-51.990,-178.021,5.831,148.444
C08096=1220.594,147.010,-51.970,-178.024,5.830,148.445
C08097=1220.599,146.760,-51.948,-178.026,5.829,148.445
C08098=1220.604,146.511,-51.927,-178.030,5.828,148.446
C08099=1220.608,146.263,-51.906,-178.032,5.827,148.446
C08100=1220.613,146.014,-51.885,-178.034,5.825,148.447
C08101=1220.618,145.765,-51.865,-178.037,5.824,148.447
C08102=1220.623,145.515,-51.844,-178.040,5.822,148.448
C08103=1220.628,145.267,-51.822,-178.042,5.822,148.448
C08104=1220.632,145.017,-51.802,-178.045,5.820,148.449
C08105=1220.637,144.768,-51.781,-178.047,5.819,148.449
C08106=1220.641,144.519,-51.760,-178.050,5.817,148.450
C08107=1220.646,144.270,-51.739,-178.052,5.816,148.450
C08108=1220.651,144.021,-51.718,-178.055,5.815,148.451
C08109=1220.656,143.772,-51.697,-178.057,5.814,148.451
C08110=1220.660,143.523,-51.677,-178.060,5.813,148.451
C08111=1220.665,143.274,-51.656,-178.063,5.812,148.452
C08112=1220.670,143.025,-51.635,-178.065,5.811,148.452
C08113=1220.675,142.776,-51.614,-178.068,5.809,148.453
C08114=1220.679,142.526,-51.594,-178.070,5.808,148.453
C08115=1220.684,142.277,-51.573,-178.073,5.806,148.454
C08116=1220.688,142.028,-51.552,-178.075,5.806,148.454
C08117=1220.693,141.779,-51.531,-178.078,5.804,148.455
C08118=1220.698,141.530,-51.510,-178.081,5.803,148.455
C08119=1220.703,141.281,-51.489,-178.083,5.801,148.456
C08120=1220.707,141.032,-51.469,-178.086,5.801,148.456
C08121=1220.712,140.783,-51.448,-178.089,5.799,148.457
C08122=1220.717,140.534,-51.428,-178.091,5.798,148.457
C08123=1220.722,140.284,-51.407,-178.094,5.797,148.458
C08124=1220.727,140.035,-51.386,-178.096,5.796,148.458
C08125=1220.731,139.787,-51.366,-178.099,5.795,148.459
C08126=1220.736,139.537,-51.345,-178.101,5.793,148.459
C08127=1220.741,139.288,-51.325,-178.104,5.792,148.460
C08128=1220.746,139.039,-51.304,-178.107,5.791,148.460
C08129=1220.750,138.790,-51.283,-178.109,5.790,148.461
C08130=1220.755,138.541,-51.262,-178.112,5.788,148.461
C08131=1220.760,138.292,-51.242,-178.114,5.787,148.462
C08132=1220.764,138.043,-51.222,-178.117,5.786,148.462
C08133=1220.769,137.794,-51.201,-178.119,5.785,148.463
C08134=1220.774,137.545,-51.180,-178.122,5.784,148.463
C08135=1220.779,137.295,-51.161,-178.124,5.782,148.464
C08136=1220.784,137.046,-51.140,-178.127,5.781,148.464
C08137=1220.788,136.797,-51.119,-178.130,5.780,148.465
C08138=1220.793,136.548,-51.099,-178.132,5.779,148.465
C08139=1220.798,136.299,-51.078,-178.135,5.778,148.466
C08140=1220.802,136.050,-51.058,-178.137,5.777,148.466
C08141=1220.807,135.801,-51.037,-178.140,5.776,148.467
C08142=1220.812,135.552,-51.016,-178.142,5.774,148.467
C08143=1220.817,135.302,-50.997,-178.145,5.774,148.468
C08144=1220.821,135.053,-50.976,-178.148,5.772,148.468
C08145=1220.826,134.804,-50.955,-178.150,5.771,148.469
C08146=1220.831,134.555,-50.935,-178.153,5.769,148.469
C08147=1220.835,134.306,-50.914,-178.155,5.768,148.469
C08148=1220.841,134.056,-50.894,-178.158,5.768,148.470
C08149=1220.845,133.788,-50.872,-178.161,5.766,148.471
C08150=1220.851,133.519,-50.851,-178.164,5.764,148.471
C08151=1220.856,133.251,-50.828,-178.166,5.764,148.472
C08152=1220.861,132.982,-50.807,-178.169,5.762,148.472
C08153=1220.866,132.733,-50.787,-178.171,5.761,148.473
C08154=1220.871,132.484,-50.766,-178.174,5.760,148.473
C08155=1220.875,132.235,-50.746,-178.177,5.759,148.474
C08156=1220.880,131.985,-50.726,-178.179,5.758,148.474
C08157=1220.884,131.736,-50.706,-178.182,5.757,148.475
C08158=1220.890,131.487,-50.685,-178.184,5.756,148.475
C08159=1220.894,131.238,-50.665,-178.187,5.754,148.476
C08160=1220.899,130.989,-50.645,-178.189,5.753,148.476
C08161=1220.904,130.740,-50.625,-178.192,5.752,148.477
C08162=1220.908,130.491,-50.605,-178.195,5.751,148.477
C08163=1220.914,130.242,-50.584,-178.197,5.750,148.478
C08164=1220.918,129.993,-50.564,-178.200,5.748,148.478
C08165=1220.923,129.743,-50.544,-178.203,5.748,148.479
C08166=1220.927,129.494,-50.523,-178.205,5.747,148.479
C08167=1220.932,129.244,-50.504,-178.208,5.745,148.480
C08168=1220.937,128.996,-50.484,-178.210,5.744,148.480
C08169=1220.941,128.747,-50.463,-178.213,5.743,148.481
C08170=1220.947,128.497,-50.443,-178.215,5.742,148.481
C08171=1220.951,128.248,-50.423,-178.218,5.741,148.482
C08172=1220.956,127.999,-50.403,-178.220,5.739,148.482
C08173=1220.961,127.750,-50.383,-178.223,5.739,148.483
C08174=1220.965,127.500,-50.363,-178.225,5.738,148.483
C08175=1220.970,127.252,-50.343,-178.228,5.736,148.484
C08176=1220.975,127.003,-50.323,-178.231,5.735,148.484
C08177=1220.980,126.754,-50.303,-178.234,5.734,148.485
C08178=1220.984,126.504,-50.283,-178.236,5.733,148.485
C08179=1220.989,126.255,-50.263,-178.238,5.732,148.486
C08180=1220.994,126.006,-50.244,-178.241,5.731,148.486
C08181=1220.999,125.757,-50.223,-178.244,5.730,148.487
C08182=1221.004,125.507,-50.203,-178.246,5.729,148.487
C08183=1221.008,125.258,-50.183,-178.249,5.728,148.488
C08184=1221.013,125.009,-50.163,-178.251,5.727,148.489
C08185=1221.018,124.761,-50.143,-178.254,5.725,148.489
C08186=1221.023,124.511,-50.123,-178.256,5.724,148.490
C08187=1221.028,124.261,-50.104,-178.259,5.724,148.490
C08188=1221.032,124.013,-50.083,-178.262,5.722,148.491
C08189=1221.037,123.764,-50.064,-178.264,5.721,148.491
C08190=1221.042,123.515,-50.044,-178.266,5.720,148.492
C08191=1221.047,123.265,-50.024,-178.270,5.719,148.492
C08192=1221.051,123.016,-50.004,-178.272,5.718,148.493
C08193=1221.056,122.767,-49.984,-178.274,5.717,148.493
C08194=1221.061,122.518,-49.965,-178.277,5.715,148.494
C08195=1221.066,122.268,-49.945,-178.280,5.715,148.494
C08196=1221.070,122.019,-49.925,-178.282,5.714,148.495
C08197=1221.076,121.770,-49.905,-178.285,5.712,148.495
C08198=1221.080,121.521,-49.886,-178.287,5.711,148.496
C08199=1221.084,121.272,-49.866,-178.290,5.711,148.496
C08200=1221.089,121.023,-49.846,-178.293,5.709,148.497
C08201=1221.094,120.774,-49.827,-178.295,5.708,148.497
C08202=1221.099,120.524,-49.807,-178.297,5.708,148.498
C08203=1221.103,120.275,-49.787,-178.300,5.706,148.498
C08204=1221.109,120.026,-49.768,-178.303,5.705,148.499
C08205=1221.113,119.777,-49.748,-178.305,5.704,148.499
C08206=1221.118,119.527,-49.728,-178.308,5.703,148.500
C08207=1221.123,119.278,-49.708,-178.310,5.702,148.501
C08208=1221.128,119.029,-49.689,-178.313,5.701,148.501
C08209=1221.133,118.780,-49.669,-178.315,5.699,148.502
C08210=1221.137,118.531,-49.650,-178.318,5.699,148.502
C08211=1221.142,118.282,-49.631,-178.320,5.698,148.503
C08212=1221.147,118.033,-49.610,-178.323,5.696,148.503
C08213=1221.151,117.783,-49.591,-178.326,5.696,148.504
C08214=1221.157,117.534,-49.571,-178.328,5.695,148.504
C08215=1221.161,117.285,-49.552,-178.331,5.693,148.505
C08216=1221.166,117.035,-49.532,-178.333,5.692,148.505
C08217=1221.171,116.787,-49.513,-178.336,5.692,148.506
C08218=1221.175,116.537,-49.494,-178.339,5.690,148.506
C08219=1221.181,116.288,-49.475,-178.341,5.689,148.507
C08220=1221.185,116.039,-49.454,-178.343,5.688,148.507
C08221=1221.190,115.790,-49.435,-178.347,5.687,148.508
C08222=1221.195,115.541,-49.416,-178.349,5.686,148.509
C08223=1221.199,115.292,-49.396,-178.351,5.685,148.509
C08224=1221.204,115.042,-49.377,-178.354,5.685,148.510
C08225=1221.209,114.793,-49.357,-178.357,5.683,148.510
C08226=1221.214,114.544,-49.338,-178.359,5.682,148.511
C08227=1221.219,114.295,-49.319,-178.361,5.681,148.511
C08228=1221.224,114.045,-49.299,-178.365,5.680,148.512
C08229=1221.228,113.796,-49.280,-178.367,5.679,148.512
C08230=1221.234,113.547,-49.260,-178.369,5.678,148.513
C08231=1221.238,113.298,-49.241,-178.372,5.677,148.513
C08232=1221.243,113.049,-49.222,-178.375,5.676,148.514
C08233=1221.248,112.799,-49.202,-178.377,5.675,148.515
C08234=1221.252,112.550,-49.183,-178.379,5.675,148.515
C08235=1221.257,112.301,-49.164,-178.382,5.673,148.516
C08236=1221.262,112.052,-49.144,-178.385,5.672,148.516
C08237=1221.267,111.803,-49.125,-178.387,5.671,148.517
C08238=1221.271,111.553,-49.106,-178.390,5.670,148.517
C08239=1221.276,111.305,-49.087,-178.393,5.669,148.518
C08240=1221.281,111.055,-49.067,-178.395,5.668,148.518
C08241=1221.286,110.805,-49.049,-178.397,5.668,148.519
C08242=1221.291,110.556,-49.029,-178.400,5.666,148.519
C08243=1221.296,110.307,-49.010,-178.403,5.665,148.520
C08244=1221.300,110.058,-48.991,-178.405,5.665,148.520
C08245=1221.305,109.809,-48.971,-178.408,5.663,148.521
C08246=1221.310,109.560,-48.952,-178.410,5.662,148.521
C08247=1221.314,109.310,-48.933,-178.413,5.662,148.522
C08248=1221.320,109.062,-48.914,-178.416,5.661,148.523
C08249=1221.325,108.811,-48.895,-178.418,5.659,148.523
C08250=1221.329,108.563,-48.876,-178.421,5.659,148.524
C08251=1221.334,108.313,-48.856,-178.423,5.658,148.524
C08252=1221.339,108.065,-48.838,-178.426,5.657,148.525
C08253=1221.344,107.796,-48.817,-178.429,5.656,148.525
C08254=1221.349,107.528,-48.797,-178.432,5.655,148.526
C08255=1221.354,107.259,-48.775,-178.434,5.653,148.526
C08256=1221.360,106.990,-48.755,-178.437,5.653,148.527
C08257=1221.364,106.741,-48.736,-178.439,5.652,148.528
C08258=1221.369,106.492,-48.717,-178.442,5.650,148.528
C08259=1221.373,106.243,-48.698,-178.445,5.650,148.529
C08260=1221.379,105.993,-48.680,-178.447,5.649,148.529
C08261=1221.383,105.744,-48.660,-178.449,5.648,148.530
C08262=1221.388,105.495,-48.641,-178.453,5.647,148.531
C08263=1221.393,105.246,-48.621,-178.455,5.646,148.531
C08264=1221.398,104.997,-48.604,-178.457,5.645,148.532
C08265=1221.403,104.747,-48.584,-178.460,5.644,148.532
C08266=1221.408,104.498,-48.565,-178.463,5.643,148.533
C08267=1221.413,104.249,-48.547,-178.465,5.642,148.533
C08268=1221.417,104.000,-48.528,-178.468,5.641,148.534
C08269=1221.422,103.751,-48.508,-178.470,5.640,148.534
C08270=1221.427,103.501,-48.490,-178.473,5.639,148.535
C08271=1221.432,103.252,-48.471,-178.475,5.638,148.535
C08272=1221.436,103.002,-48.452,-178.478,5.637,148.536
C08273=1221.442,102.753,-48.433,-178.481,5.637,148.537
C08274=1221.446,102.505,-48.414,-178.483,5.635,148.537
C08275=1221.451,102.255,-48.396,-178.486,5.634,148.538
C08276=1221.456,102.006,-48.377,-178.489,5.634,148.538
C08277=1221.460,101.756,-48.358,-178.491,5.633,148.539
C08278=1221.466,101.507,-48.339,-178.494,5.631,148.539
C08279=1221.470,101.257,-48.321,-178.496,5.631,148.540
C08280=1221.475,101.009,-48.301,-178.499,5.630,148.540
C08281=1221.480,100.760,-48.283,-178.501,5.629,148.541
C08282=1221.485,100.510,-48.264,-178.503,5.628,148.542
C08283=1221.490,100.261,-48.245,-178.507,5.627,148.542
C08284=1221.495,100.012,-48.227,-178.509,5.626,148.543
C08285=1221.499,99.763,-48.207,-178.511,5.625,148.543
C08286=1221.504,99.513,-48.189,-178.514,5.625,148.544
C08287=1221.508,99.264,-48.170,-178.517,5.623,148.545
C08288=1221.514,99.015,-48.152,-178.519,5.622,148.545
C08289=1221.518,98.766,-48.133,-178.522,5.622,148.546
C08290=1221.524,98.516,-48.114,-178.524,5.621,148.546
C08291=1221.528,98.267,-48.096,-178.527,5.620,148.547
C08292=1221.533,98.018,-48.077,-178.530,5.619,148.547
C08293=1221.538,97.768,-48.059,-178.532,5.618,148.548
C08294=1221.543,97.519,-48.040,-178.534,5.617,148.548
C08295=1221.548,97.270,-48.022,-178.537,5.617,148.549
C08296=1221.552,97.021,-48.002,-178.539,5.616,148.549
C08297=1221.557,96.771,-47.984,-178.542,5.614,148.550
C08298=1221.562,96.522,-47.966,-178.545,5.614,148.551
C08299=1221.567,96.273,-47.947,-178.547,5.613,148.551
C08300=1221.572,96.024,-47.929,-178.550,5.612,148.552
C08301=1221.577,95.774,-47.911,-178.552,5.612,148.552
C08302=1221.581,95.525,-47.891,-178.555,5.610,148.553
C08303=1221.586,95.276,-47.873,-178.558,5.609,148.554
C08304=1221.591,95.026,-47.855,-178.560,5.609,148.554
C08305=1221.596,94.778,-47.836,-178.562,5.608,148.555
C08306=1221.601,94.528,-47.817,-178.565,5.607,148.555
C08307=1221.606,94.279,-47.799,-178.568,5.606,148.556
C08308=1221.610,94.030,-47.781,-178.570,5.605,148.556
C08309=1221.615,93.780,-47.762,-178.573,5.604,148.557
C08310=1221.620,93.531,-47.744,-178.576,5.603,148.558
C08311=1221.625,93.281,-47.726,-178.578,5.603,148.558
C08312=1221.630,93.033,-47.707,-178.581,5.601,148.559
C08313=1221.634,92.783,-47.689,-178.584,5.600,148.559
C08314=1221.639,92.534,-47.671,-178.586,5.600,148.560
C08315=1221.645,92.284,-47.652,-178.588,5.599,148.560
C08316=1221.649,92.036,-47.633,-178.591,5.598,148.561
C08317=1221.654,91.786,-47.615,-178.594,5.598,148.562
C08318=1221.659,91.537,-47.597,-178.596,5.596,148.562
C08319=1221.664,91.288,-47.579,-178.599,5.595,148.563
C08320=1221.669,91.038,-47.561,-178.601,5.595,148.563
C08321=1221.673,90.789,-47.542,-178.604,5.594,148.564
C08322=1221.678,90.540,-47.524,-178.606,5.593,148.564
C08323=1221.683,90.290,-47.506,-178.609,5.593,148.565
C08324=1221.688,90.041,-47.488,-178.612,5.591,148.566
C08325=1221.692,89.791,-47.469,-178.614,5.590,148.566
C08326=1221.698,89.542,-47.451,-178.617,5.590,148.567
C08327=1221.703,89.293,-47.433,-178.619,5.589,148.567
C08328=1221.707,89.044,-47.414,-178.622,5.588,148.568
C08329=1221.712,88.795,-47.396,-178.624,5.588,148.569
C08330=1221.717,88.545,-47.378,-178.627,5.586,148.569
C08331=1221.722,88.296,-47.360,-178.630,5.585,148.570
C08332=1221.726,88.047,-47.342,-178.632,5.585,148.570
C08333=1221.731,87.798,-47.324,-178.635,5.584,148.571
C08334=1221.737,87.548,-47.305,-178.637,5.583,148.571
C08335=1221.742,87.299,-47.287,-178.640,5.582,148.572
C08336=1221.746,87.049,-47.269,-178.642,5.582,148.573
C08337=1221.751,86.800,-47.251,-178.645,5.580,148.573
C08338=1221.756,86.551,-47.233,-178.647,5.580,148.574
C08339=1221.761,86.302,-47.215,-178.650,5.579,148.574
C08340=1221.766,86.052,-47.197,-178.652,5.578,148.575
C08341=1221.771,85.803,-47.179,-178.655,5.577,148.575
C08342=1221.775,85.553,-47.161,-178.657,5.577,148.576
C08343=1221.780,85.304,-47.143,-178.660,5.576,148.577
C08344=1221.785,85.055,-47.125,-178.663,5.574,148.577
C08345=1221.790,84.806,-47.107,-178.665,5.574,148.578
C08346=1221.795,84.557,-47.089,-178.668,5.573,148.579
C08347=1221.800,84.307,-47.071,-178.670,5.572,148.579
C08348=1221.805,84.058,-47.053,-178.673,5.572,148.580
C08349=1221.810,83.809,-47.035,-178.675,5.571,148.580
C08350=1221.814,83.559,-47.016,-178.678,5.571,148.581
C08351=1221.819,83.310,-46.998,-178.681,5.569,148.581
C08352=1221.824,83.061,-46.980,-178.683,5.568,148.582
C08353=1221.829,82.811,-46.963,-178.686,5.568,148.583
C08354=1221.834,82.562,-46.945,-178.688,5.567,148.583
C08355=1221.839,82.313,-46.927,-178.691,5.566,148.584
C08356=1221.844,82.064,-46.909,-178.693,5.566,148.584
C08357=1221.849,81.795,-46.890,-178.696,5.565,148.585
C08358=1221.854,81.527,-46.870,-178.699,5.564,148.586
C08359=1221.859,81.258,-46.852,-178.702,5.563,148.586
C08360=1221.864,80.990,-46.832,-178.704,5.562,148.587
C08361=1221.869,80.741,-46.814,-178.707,5.561,148.587
C08362=1221.874,80.492,-46.796,-178.710,5.560,148.588
C08363=1221.879,80.242,-46.779,-178.712,5.559,148.589
C08364=1221.884,79.993,-46.761,-178.715,5.559,148.589
C08365=1221.889,79.743,-46.743,-178.717,5.558,148.590
C08366=1221.894,79.494,-46.725,-178.720,5.557,148.590
C08367=1221.899,79.245,-46.707,-178.722,5.557,148.591
C08368=1221.903,78.996,-46.691,-178.725,5.556,148.592
C08369=1221.908,78.746,-46.673,-178.727,5.555,148.592
C08370=1221.913,78.497,-46.655,-178.730,5.555,148.593
C08371=1221.918,78.248,-46.637,-178.733,5.553,148.593
C08372=1221.923,77.998,-46.619,-178.735,5.552,148.594
C08373=1221.928,77.748,-46.601,-178.738,5.552,148.595
C08374=1221.933,77.499,-46.583,-178.740,5.551,148.595
C08375=1221.937,77.250,-46.566,-178.743,5.550,148.596
C08376=1221.942,77.001,-46.548,-178.745,5.550,148.596
C08377=1221.947,76.751,-46.530,-178.748,5.549,148.597
C08378=1221.952,76.502,-46.513,-178.750,5.548,148.598
C08379=1221.957,76.252,-46.495,-178.753,5.548,148.598
C08380=1221.962,76.003,-46.477,-178.755,5.547,148.599
C08381=1221.966,75.754,-46.460,-178.758,5.545,148.599
C08382=1221.971,75.505,-46.442,-178.761,5.545,148.600
C08383=1221.976,75.255,-46.424,-178.764,5.544,148.601
C08384=1221.981,75.006,-46.407,-178.766,5.543,148.601
C08385=1221.986,74.757,-46.390,-178.768,5.543,148.602
C08386=1221.991,74.507,-46.373,-178.771,5.542,148.602
C08387=1221.996,74.258,-46.355,-178.774,5.542,148.603
C08388=1222.001,74.009,-46.337,-178.776,5.541,148.604
C08389=1222.007,73.759,-46.320,-178.778,5.540,148.604
C08390=1222.011,73.511,-46.302,-178.781,5.540,148.605
C08391=1222.016,73.261,-46.285,-178.784,5.539,148.606
C08392=1222.021,73.012,-46.267,-178.786,5.538,148.606
C08393=1222.025,72.762,-46.250,-178.789,5.537,148.607
C08394=1222.030,72.513,-46.232,-178.792,5.536,148.607
C08395=1222.035,72.263,-46.215,-178.794,5.535,148.608
C08396=1222.040,72.014,-46.197,-178.797,5.535,148.609
C08397=1222.045,71.765,-46.181,-178.799,5.534,148.609
C08398=1222.050,71.515,-46.163,-178.802,5.533,148.610
C08399=1222.055,71.266,-46.145,-178.804,5.533,148.610
C08400=1222.059,71.017,-46.128,-178.807,5.532,148.611
C08401=1222.064,70.767,-46.111,-178.809,5.531,148.611
C08402=1222.069,70.518,-46.093,-178.812,5.531,148.612
C08403=1222.074,70.269,-46.076,-178.814,5.530,148.613
C08404=1222.079,70.020,-46.058,-178.817,5.530,148.613
C08405=1222.084,69.770,-46.041,-178.820,5.529,148.614
C08406=1222.089,69.521,-46.024,-178.822,5.528,148.614
C08407=1222.094,69.271,-46.006,-178.824,5.527,148.615
C08408=1222.099,69.022,-45.989,-178.827,5.526,148.616
C08409=1222.103,68.773,-45.972,-178.830,5.525,148.616
C08410=1222.108,68.523,-45.955,-178.832,5.525,148.617
C08411=1222.113,68.274,-45.937,-178.835,5.524,148.618
C08412=1222.118,68.024,-45.920,-178.838,5.523,148.618
C08413=1222.124,67.775,-45.903,-178.840,5.523,148.619
C08414=1222.128,67.526,-45.886,-178.843,5.522,148.620
C08415=1222.133,67.276,-45.868,-178.845,5.521,148.620
C08416=1222.138,67.027,-45.851,-178.848,5.521,148.621
C08417=1222.142,66.778,-45.834,-178.850,5.520,148.621
C08418=1222.148,66.528,-45.816,-178.853,5.520,148.622
C08419=1222.152,66.279,-45.800,-178.855,5.519,148.622
C08420=1222.158,66.030,-45.782,-178.858,5.518,148.623
C08421=1222.162,65.781,-45.765,-178.860,5.517,148.624
C08422=1222.167,65.531,-45.748,-178.863,5.517,148.624
C08423=1222.172,65.281,-45.732,-178.865,5.516,148.625
C08424=1222.177,65.032,-45.714,-178.868,5.515,148.625
C08425=1222.182,64.782,-45.696,-178.870,5.515,148.626
C08426=1222.187,64.534,-45.680,-178.873,5.514,148.627
C08427=1222.192,64.284,-45.663,-178.876,5.514,148.627
C08428=1222.196,64.035,-45.645,-178.878,5.513,148.628
C08429=1222.202,63.785,-45.628,-178.880,5.512,148.629
C08430=1222.206,63.536,-45.611,-178.883,5.512,148.629
C08431=1222.212,63.286,-45.595,-178.886,5.511,148.630
C08432=1222.216,63.038,-45.577,-178.888,5.510,148.631
C08433=1222.221,62.788,-45.560,-178.891,5.509,148.631
C08434=1222.226,62.538,-45.543,-178.894,5.508,148.632
C08435=1222.231,62.289,-45.526,-178.896,5.508,148.632
C08436=1222.236,62.040,-45.510,-178.899,5.507,148.633
C08437=1222.241,61.790,-45.492,-178.901,5.506,148.634
C08438=1222.246,61.541,-45.475,-178.904,5.506,148.634
C08439=1222.250,61.292,-45.458,-178.906,5.505,148.635
C08440=1222.256,61.043,-45.441,-178.909,5.504,148.635
C08441=1222.260,60.793,-45.425,-178.911,5.504,148.636
C08442=1222.266,60.543,-45.407,-178.914,5.503,148.637
C08443=1222.270,60.294,-45.391,-178.917,5.503,148.637
C08444=1222.276,60.045,-45.374,-178.919,5.502,148.638
C08445=1222.280,59.795,-45.357,-178.921,5.501,148.639
C08446=1222.285,59.546,-45.341,-178.924,5.501,148.639
C08447=1222.290,59.297,-45.323,-178.927,5.500,148.640
C08448=1222.295,59.048,-45.306,-178.929,5.499,148.640
C08449=1222.300,58.798,-45.289,-178.932,5.499,148.641
C08450=1222.304,58.548,-45.272,-178.934,5.498,148.642
C08451=1222.309,58.299,-45.256,-178.937,5.497,148.642
C08452=1222.315,58.050,-45.239,-178.939,5.497,148.643
C08453=1222.319,57.800,-45.222,-178.942,5.496,148.644
C08454=1222.324,57.551,-45.205,-178.945,5.496,148.644
C08455=1222.330,57.302,-45.189,-178.947,5.495,148.645
C08456=1222.334,57.052,-45.172,-178.949,5.494,148.645
C08457=1222.339,56.803,-45.155,-178.952,5.494,148.646
C08458=1222.344,56.554,-45.138,-178.955,5.493,148.647
C08459=1222.349,56.304,-45.122,-178.957,5.492,148.647
C08460=1222.354,56.054,-45.104,-178.960,5.492,148.648
C08461=1222.360,55.786,-45.087,-178.963,5.491,148.649
C08462=1222.364,55.517,-45.069,-178.965,5.491,148.649
C08463=1222.370,55.249,-45.051,-178.968,5.490,148.650
C08464=1222.375,54.981,-45.033,-178.971,5.490,148.651
C08465=1222.380,54.732,-45.017,-178.973,5.489,148.651
C08466=1222.385,54.482,-44.999,-178.975,5.488,148.652
C08467=1222.390,54.233,-44.983,-178.978,5.488,148.652
C08468=1222.395,53.983,-44.967,-178.981,5.487,148.653
C08469=1222.400,53.733,-44.950,-178.983,5.486,148.654
C08470=1222.405,53.484,-44.933,-178.986,5.486,148.654
C08471=1222.410,53.235,-44.917,-178.989,5.485,148.655
C08472=1222.414,52.986,-44.900,-178.991,5.485,148.656
C08473=1222.420,52.736,-44.883,-178.993,5.484,148.656
C08474=1222.425,52.487,-44.867,-178.996,5.483,148.657
C08475=1222.429,52.237,-44.851,-178.999,5.483,148.658
C08476=1222.434,51.988,-44.834,-179.001,5.482,148.658
C08477=1222.440,51.738,-44.817,-179.004,5.482,148.659
C08478=1222.444,51.489,-44.800,-179.006,5.481,148.660
C08479=1222.449,51.240,-44.784,-179.009,5.480,148.660
C08480=1222.454,50.990,-44.768,-179.011,5.480,148.661
C08481=1222.459,50.741,-44.751,-179.014,5.479,148.661
C08482=1222.464,50.491,-44.735,-179.017,5.478,148.662
C08483=1222.469,50.242,-44.718,-179.019,5.478,148.663
C08484=1222.474,49.993,-44.702,-179.022,5.477,148.663
C08485=1222.479,49.743,-44.686,-179.024,5.476,148.664
C08486=1222.483,49.494,-44.669,-179.027,5.476,148.664
C08487=1222.488,49.245,-44.653,-179.029,5.475,148.665
C08488=1222.493,48.995,-44.635,-179.032,5.475,148.666
C08489=1222.499,48.746,-44.620,-179.035,5.474,148.667
C08490=1222.503,48.496,-44.603,-179.037,5.474,148.667
C08491=1222.508,48.247,-44.586,-179.040,5.473,148.668
C08492=1222.513,47.997,-44.571,-179.042,5.472,148.668
C08493=1222.518,47.748,-44.554,-179.044,5.472,148.669
C08494=1222.523,47.499,-44.538,-179.047,5.472,148.670
C08495=1222.528,47.249,-44.521,-179.049,5.471,148.670
C08496=1222.533,47.000,-44.505,-179.052,5.471,148.671
C08497=1222.538,46.750,-44.488,-179.055,5.470,148.672
C08498=1222.543,46.501,-44.473,-179.057,5.470,148.672
C08499=1222.548,46.251,-44.456,-179.059,5.469,148.673
C08500=1222.553,46.003,-44.440,-179.062,5.468,148.673
C08501=1222.558,45.753,-44.424,-179.065,5.468,148.674
C08502=1222.562,45.503,-44.407,-179.067,5.467,148.675
C08503=1222.567,45.254,-44.392,-179.070,5.466,148.675
C08504=1222.572,45.004,-44.375,-179.073,5.466,148.676
C08505=1222.578,44.755,-44.358,-179.075,5.465,148.677
C08506=1222.583,44.505,-44.342,-179.078,5.465,148.677
C08507=1222.588,44.256,-44.326,-179.080,5.464,148.678
C08508=1222.592,44.006,-44.310,-179.083,5.463,148.679
C08509=1222.597,43.757,-44.294,-179.085,5.463,148.679
C08510=1222.602,43.507,-44.278,-179.088,5.462,148.680
C08511=1222.607,43.258,-44.261,-179.090,5.462,148.681
C08512=1222.612,43.008,-44.245,-179.093,5.462,148.681
C08513=1222.617,42.760,-44.229,-179.095,5.461,148.682
C08514=1222.622,42.509,-44.213,-179.097,5.460,148.682
C08515=1222.627,42.261,-44.197,-179.100,5.460,148.683
C08516=1222.632,42.011,-44.181,-179.103,5.459,148.684
C08517=1222.637,41.762,-44.164,-179.105,5.459,148.684
C08518=1222.642,41.512,-44.149,-179.108,5.458,148.685
C08519=1222.647,41.263,-44.132,-179.111,5.458,148.686
C08520=1222.652,41.013,-44.117,-179.113,5.457,148.686
C08521=1222.657,40.764,-44.100,-179.116,5.457,148.687
C08522=1222.662,40.515,-44.084,-179.118,5.456,148.688
C08523=1222.667,40.265,-44.068,-179.121,5.455,148.688
C08524=1222.672,40.016,-44.052,-179.123,5.455,148.689
C08525=1222.677,39.766,-44.036,-179.125,5.455,148.690
C08526=1222.682,39.517,-44.020,-179.128,5.454,148.690
C08527=1222.686,39.268,-44.005,-179.131,5.454,148.691
C08528=1222.691,39.018,-43.988,-179.133,5.453,148.692
C08529=1222.696,38.769,-43.973,-179.136,5.453,148.692
C08530=1222.701,38.519,-43.957,-179.139,5.452,148.693
C08531=1222.706,38.270,-43.940,-179.141,5.451,148.693
C08532=1222.711,38.020,-43.924,-179.143,5.451,148.694
C08533=1222.716,37.770,-43.909,-179.146,5.450,148.695
C08534=1222.721,37.522,-43.893,-179.149,5.449,148.695
C08535=1222.726,37.272,-43.877,-179.151,5.449,148.696
C08536=1222.732,37.022,-43.861,-179.153,5.449,148.697
C08537=1222.736,36.773,-43.844,-179.156,5.449,148.697
C08538=1222.741,36.524,-43.829,-179.159,5.448,148.698
C08539=1222.746,36.274,-43.814,-179.161,5.447,148.699
C08540=1222.751,36.025,-43.797,-179.163,5.447,148.699
C08541=1222.756,35.775,-43.781,-179.166,5.446,148.700
C08542=1222.761,35.526,-43.766,-179.169,5.445,148.701
C08543=1222.766,35.276,-43.750,-179.171,5.445,148.701
C08544=1222.771,35.027,-43.734,-179.174,5.444,148.702
C08545=1222.775,34.777,-43.718,-179.177,5.444,148.703
C08546=1222.781,34.528,-43.703,-179.179,5.444,148.703
C08547=1222.786,34.278,-43.687,-179.181,5.444,148.704
C08548=1222.791,34.029,-43.670,-179.184,5.443,148.705
C08549=1222.796,33.780,-43.655,-179.187,5.442,148.705
C08550=1222.801,33.530,-43.640,-179.189,5.442,148.706
C08551=1222.805,33.280,-43.624,-179.191,5.441,148.706
C08552=1222.810,33.032,-43.608,-179.194,5.440,148.707
C08553=1222.816,32.782,-43.592,-179.197,5.440,148.708
C08554=1222.821,32.532,-43.576,-179.199,5.439,148.708
C08555=1222.825,32.283,-43.561,-179.201,5.440,148.709
C08556=1222.831,32.034,-43.545,-179.204,5.439,148.710
C08557=1222.835,31.783,-43.530,-179.207,5.439,148.711
C08558=1222.841,31.535,-43.513,-179.209,5.438,148.711
C08559=1222.845,31.286,-43.498,-179.212,5.437,148.712
C08560=1222.850,31.035,-43.482,-179.214,5.437,148.712
C08561=1222.855,30.786,-43.467,-179.217,5.436,148.713
C08562=1222.861,30.537,-43.451,-179.219,5.435,148.714
C08563=1222.865,30.288,-43.436,-179.221,5.436,148.714
C08564=1222.870,30.037,-43.420,-179.224,5.435,148.715
C08565=1222.876,29.769,-43.403,-179.227,5.435,148.716
C08566=1222.881,29.501,-43.386,-179.229,5.434,148.716
C08567=1222.886,29.232,-43.370,-179.232,5.434,148.717
C08568=1222.892,28.963,-43.353,-179.235,5.433,148.718
C08569=1222.897,28.713,-43.337,-179.238,5.433,148.719
C08570=1222.902,28.464,-43.322,-179.240,5.432,148.719
C08571=1222.907,28.215,-43.307,-179.243,5.431,148.720
C08572=1222.912,27.965,-43.291,-179.245,5.431,148.720
C08573=1222.917,27.716,-43.275,-179.248,5.430,148.721
C08574=1222.921,27.467,-43.260,-179.251,5.430,148.722
C08575=1222.927,27.217,-43.244,-179.253,5.430,148.722
C08576=1222.932,26.968,-43.228,-179.255,5.429,148.723
C08577=1222.936,26.717,-43.214,-179.258,5.429,148.724
C08578=1222.942,26.468,-43.198,-179.261,5.428,148.725
C08579=1222.946,26.219,-43.183,-179.263,5.428,148.725
C08580=1222.952,25.970,-43.168,-179.266,5.427,148.726
C08581=1222.957,25.719,-43.152,-179.268,5.427,148.727
C08582=1222.961,25.470,-43.137,-179.270,5.427,148.727
C08583=1222.967,25.221,-43.121,-179.273,5.426,148.728
C08584=1222.972,24.972,-43.105,-179.275,5.426,148.728
C08585=1222.977,24.722,-43.090,-179.278,5.425,148.729
C08586=1222.981,24.472,-43.075,-179.281,5.425,148.730
C08587=1222.986,24.223,-43.060,-179.283,5.424,148.730
C08588=1222.992,23.974,-43.044,-179.286,5.423,148.731
C08589=1222.997,23.724,-43.028,-179.288,5.424,148.732
C08590=1223.001,23.475,-43.013,-179.291,5.423,148.732
C08591=1223.007,23.225,-42.998,-179.293,5.423,148.733
C08592=1223.011,22.976,-42.983,-179.296,5.422,148.734
C08593=1223.017,22.726,-42.968,-179.299,5.422,148.735
C08594=1223.021,22.477,-42.953,-179.301,5.421,148.735
C08595=1223.027,22.228,-42.937,-179.303,5.421,148.736
C08596=1223.031,21.978,-42.922,-179.305,5.420,148.736
C08597=1223.036,21.728,-42.906,-179.308,5.420,148.737
C08598=1223.041,21.479,-42.892,-179.311,5.419,148.738
C08599=1223.046,21.229,-42.876,-179.313,5.419,148.738
C08600=1223.052,20.980,-42.861,-179.316,5.418,148.739
C08601=1223.057,20.731,-42.846,-179.318,5.419,148.740
C08602=1223.061,20.481,-42.830,-179.321,5.418,148.740
C08603=1223.066,20.231,-42.815,-179.323,5.417,148.741
C08604=1223.072,19.982,-42.800,-179.326,5.417,148.742
C08605=1223.076,19.733,-42.785,-179.329,5.416,148.742
C08606=1223.082,19.483,-42.769,-179.331,5.416,148.743
C08607=1223.087,19.233,-42.755,-179.333,5.416,148.744
C08608=1223.091,18.984,-42.740,-179.336,5.416,148.745
C08609=1223.096,18.734,-42.724,-179.339,5.415,148.745
C08610=1223.101,18.485,-42.709,-179.341,5.414,148.746
C08611=1223.106,18.235,-42.694,-179.344,5.414,148.746
C08612=1223.111,17.986,-42.679,-179.346,5.413,148.747
C08613=1223.116,17.737,-42.664,-179.348,5.413,148.748
C08614=1223.121,17.487,-42.649,-179.351,5.413,148.748
C08615=1223.127,17.238,-42.634,-179.354,5.412,148.749
C08616=1223.131,16.988,-42.619,-179.356,5.412,148.750
C08617=1223.136,16.739,-42.604,-179.359,5.411,148.750
C08618=1223.141,16.489,-42.588,-179.361,5.411,148.751
C08619=1223.146,16.240,-42.573,-179.364,5.411,148.752
C08620=1223.152,15.990,-42.559,-179.366,5.410,148.752
C08621=1223.156,15.740,-42.544,-179.369,5.410,148.753
C08622=1223.161,15.491,-42.529,-179.372,5.409,148.754
C08623=1223.167,15.241,-42.514,-179.374,5.409,148.755
C08624=1223.171,14.992,-42.499,-179.376,5.409,148.755
C08625=1223.177,14.742,-42.484,-179.379,5.409,148.756
C08626=1223.182,14.493,-42.469,-179.382,5.408,148.757
C08627=1223.186,14.244,-42.454,-179.384,5.407,148.757
C08628=1223.192,13.994,-42.439,-179.386,5.407,148.758
C08629=1223.197,13.745,-42.424,-179.388,5.407,148.758
C08630=1223.201,13.495,-42.410,-179.391,5.406,148.759
C08631=1223.207,13.246,-42.394,-179.394,5.406,148.760
C08632=1223.212,12.996,-42.380,-179.396,5.405,148.760
C08633=1223.216,12.747,-42.365,-179.399,5.405,148.761
C08634=1223.221,12.497,-42.349,-179.401,5.405,148.762
C08635=1223.226,12.247,-42.335,-179.404,5.405,148.763
C08636=1223.231,11.998,-42.320,-179.406,5.404,148.763
C08637=1223.237,11.748,-42.305,-179.409,5.403,148.764
C08638=1223.241,11.499,-42.290,-179.412,5.403,148.765
C08639=1223.246,11.249,-42.275,-179.414,5.403,148.765
C08640=1223.252,11.000,-42.260,-179.416,5.403,148.766
C08641=1223.256,10.750,-42.246,-179.419,5.402,148.767
C08642=1223.261,10.500,-42.231,-179.422,5.402,148.767
C08643=1223.266,10.251,-42.216,-179.424,5.401,148.768
C08644=1223.272,10.001,-42.201,-179.426,5.401,148.769
C08645=1223.276,9.752,-42.186,-179.429,5.401,148.769
C08646=1223.281,9.503,-42.172,-179.432,5.400,148.770
C08647=1223.286,9.253,-42.157,-179.434,5.400,148.771
C08648=1223.292,9.003,-42.142,-179.437,5.399,148.771
C08649=1223.296,8.754,-42.127,-179.439,5.399,148.772
C08650=1223.301,8.505,-42.113,-179.441,5.399,148.773
C08651=1223.306,8.255,-42.099,-179.444,5.398,148.773
C08652=1223.312,8.005,-42.083,-179.447,5.398,148.774
C08653=1223.317,7.756,-42.069,-179.449,5.397,148.775
C08654=1223.322,7.507,-42.054,-179.451,5.397,148.775
C08655=1223.327,7.258,-42.040,-179.454,5.397,148.776
C08656=1223.333,7.008,-42.025,-179.457,5.396,148.777
C08657=1223.337,6.759,-42.010,-179.459,5.396,148.777
C08658=1223.342,6.509,-41.996,-179.461,5.396,148.778
C08659=1223.347,6.259,-41.982,-179.464,5.396,148.779
C08660=1223.352,6.010,-41.967,-179.467,5.395,148.779
C08661=1223.357,5.760,-41.952,-179.469,5.395,148.780
C08662=1223.362,5.510,-41.937,-179.472,5.394,148.781
C08663=1223.367,5.261,-41.922,-179.474,5.394,148.781
C08664=1223.372,5.012,-41.908,-179.477,5.394,148.782
C08665=1223.377,4.762,-41.894,-179.479,5.393,148.783
C08666=1223.382,4.512,-41.880,-179.482,5.393,148.784
C08667=1223.387,4.263,-41.865,-179.484,5.393,148.784
C08668=1223.392,4.013,-41.850,-179.487,5.393,148.785
C08669=1223.398,3.745,-41.834,-179.489,5.392,148.786
C08670=1223.403,3.475,-41.819,-179.492,5.391,148.786
C08671=1223.409,3.207,-41.804,-179.495,5.391,148.787
C08672=1223.414,2.938,-41.788,-179.497,5.390,148.788
C08673=1223.419,2.688,-41.774,-179.500,5.390,148.788
C08674=1223.424,2.438,-41.759,-179.502,5.390,148.789
C08675=1223.429,2.189,-41.744,-179.505,5.390,148.790
C08676=1223.434,1.939,-41.730,-179.507,5.389,148.790
C08677=1223.439,1.690,-41.715,-179.510,5.389,148.791
C08678=1223.444,1.441,-41.701,-179.512,5.389,148.792
C08679=1223.449,1.191,-41.687,-179.515,5.388,148.792
C08680=1223.454,0.941,-41.673,-179.517,5.388,148.793
C08681=1223.459,0.692,-41.658,-179.520,5.387,148.794
C08682=1223.464,0.442,-41.644,-179.522,5.388,148.795
C08683=1223.469,0.193,-41.629,-179.525,5.387,148.795
C08684=1223.474,-0.057,-41.615,-179.527,5.387,148.796
C08685=1223.479,-0.306,-41.601,-179.530,5.386,148.797
C08686=1223.484,-0.556,-41.587,-179.532,5.386,148.797
C08687=1223.489,-0.805,-41.573,-179.535,5.386,148.798
C08688=1223.494,-1.055,-41.558,-179.537,5.385,148.799
C08689=1223.499,-1.304,-41.543,-179.540,5.385,148.799
C08690=1223.504,-1.554,-41.529,-179.542,5.385,148.800
C08691=1223.509,-1.803,-41.515,-179.545,5.385,148.801
C08692=1223.514,-2.053,-41.501,-179.547,5.384,148.801
C08693=1223.519,-2.302,-41.487,-179.550,5.384,148.802
C08694=1223.524,-2.552,-41.472,-179.552,5.384,148.803
C08695=1223.529,-2.802,-41.458,-179.555,5.383,148.804
C08696=1223.534,-3.052,-41.444,-179.558,5.383,148.804
C08697=1223.540,-3.301,-41.430,-179.560,5.382,148.805
C08698=1223.545,-3.550,-41.416,-179.562,5.383,148.806
C08699=1223.550,-3.800,-41.401,-179.565,5.382,148.806
C08700=1223.555,-4.050,-41.387,-179.568,5.382,148.807
C08701=1223.560,-4.299,-41.373,-179.570,5.381,148.808
C08702=1223.565,-4.548,-41.359,-179.572,5.381,148.808
C08703=1223.570,-4.798,-41.345,-179.575,5.381,148.809
C08704=1223.575,-5.048,-41.330,-179.578,5.380,148.810
C08705=1223.580,-5.297,-41.316,-179.580,5.381,148.810
C08706=1223.586,-5.546,-41.302,-179.582,5.380,148.811
C08707=1223.590,-5.796,-41.288,-179.585,5.380,148.812
C08708=1223.595,-6.046,-41.274,-179.588,5.379,148.812
C08709=1223.600,-6.296,-41.259,-179.590,5.379,148.813
C08710=1223.606,-6.545,-41.245,-179.592,5.379,148.814
C08711=1223.610,-6.794,-41.232,-179.595,5.378,148.814
C08712=1223.615,-7.044,-41.217,-179.597,5.377,148.815
C08713=1223.620,-7.293,-41.203,-179.599,5.378,148.816
C08714=1223.626,-7.542,-41.189,-179.602,5.377,148.816
C08715=1223.631,-7.793,-41.176,-179.605,5.377,148.817
C08716=1223.636,-8.043,-41.161,-179.607,5.377,148.818
C08717=1223.641,-8.292,-41.147,-179.609,5.377,148.818
C08718=1223.646,-8.541,-41.133,-179.612,5.376,148.819
C08719=1223.651,-8.791,-41.119,-179.615,5.376,148.820
C08720=1223.656,-9.040,-41.105,-179.617,5.376,148.821
C08721=1223.660,-9.290,-41.091,-179.619,5.375,148.821
C08722=1223.666,-9.539,-41.077,-179.622,5.375,148.822
C08723=1223.671,-9.789,-41.063,-179.625,5.374,148.823
C08724=1223.676,-10.039,-41.049,-179.627,5.375,148.823
C08725=1223.681,-10.288,-41.036,-179.629,5.374,148.824
C08726=1223.686,-10.538,-41.022,-179.632,5.374,148.825
C08727=1223.691,-10.787,-41.007,-179.634,5.374,148.825
C08728=1223.696,-11.038,-40.994,-179.637,5.373,148.826
C08729=1223.702,-11.287,-40.980,-179.639,5.373,148.827
C08730=1223.706,-11.536,-40.966,-179.642,5.372,148.827
C08731=1223.711,-11.786,-40.952,-179.644,5.373,148.828
C08732=1223.717,-12.035,-40.938,-179.647,5.372,148.829
C08733=1223.722,-12.285,-40.924,-179.649,5.372,148.830
C08734=1223.727,-12.535,-40.910,-179.652,5.372,148.830
C08735=1223.732,-12.783,-40.897,-179.654,5.371,148.831
C08736=1223.737,-13.033,-40.883,-179.657,5.371,148.832
C08737=1223.742,-13.283,-40.869,-179.659,5.371,148.832
C08738=1223.747,-13.532,-40.855,-179.662,5.371,148.833
C08739=1223.752,-13.782,-40.841,-179.664,5.370,148.834
C08740=1223.757,-14.032,-40.828,-179.667,5.370,148.834
C08741=1223.762,-14.281,-40.814,-179.669,5.370,148.835
C08742=1223.767,-14.531,-40.800,-179.672,5.369,148.836
C08743=1223.772,-14.781,-40.787,-179.674,5.369,148.836
C08744=1223.777,-15.030,-40.773,-179.676,5.369,148.837
C08745=1223.782,-15.280,-40.758,-179.679,5.369,148.838
C08746=1223.787,-15.529,-40.746,-179.682,5.368,148.839
C08747=1223.792,-15.779,-40.732,-179.684,5.368,148.839
C08748=1223.797,-16.028,-40.717,-179.686,5.368,148.840
C08749=1223.803,-16.278,-40.704,-179.689,5.368,148.841
C08750=1223.807,-16.527,-40.690,-179.692,5.367,148.841
C08751=1223.812,-16.777,-40.676,-179.694,5.367,148.842
C08752=1223.818,-17.027,-40.663,-179.696,5.367,148.843
C08753=1223.822,-17.276,-40.649,-179.699,5.366,148.843
C08754=1223.828,-17.526,-40.636,-179.701,5.367,148.844
C08755=1223.833,-17.776,-40.622,-179.704,5.366,148.845
C08756=1223.838,-18.025,-40.608,-179.707,5.366,148.846
C08757=1223.843,-18.275,-40.595,-179.709,5.366,148.846
C08758=1223.848,-18.524,-40.581,-179.711,5.365,148.847
C08759=1223.853,-18.774,-40.568,-179.714,5.365,148.848
C08760=1223.858,-19.023,-40.554,-179.716,5.365,148.848
C08761=1223.864,-19.273,-40.541,-179.719,5.365,148.849
C08762=1223.869,-19.522,-40.527,-179.721,5.364,148.850
C08763=1223.873,-19.772,-40.513,-179.724,5.364,148.850
C08764=1223.879,-20.021,-40.500,-179.726,5.364,148.851
C08765=1223.884,-20.271,-40.486,-179.729,5.364,148.852
C08766=1223.889,-20.521,-40.473,-179.731,5.363,148.852
C08767=1223.894,-20.770,-40.459,-179.733,5.363,148.853
C08768=1223.899,-21.020,-40.446,-179.736,5.363,148.854
C08769=1223.904,-21.269,-40.432,-179.739,5.362,148.855
C08770=1223.910,-21.519,-40.419,-179.741,5.363,148.855
C08771=1223.915,-21.769,-40.405,-179.744,5.362,148.856
C08772=1223.919,-22.018,-40.392,-179.746,5.362,148.857
C08773=1223.925,-22.287,-40.377,-179.748,5.362,148.857
C08774=1223.931,-22.557,-40.363,-179.751,5.361,148.858
C08775=1223.936,-22.826,-40.348,-179.754,5.361,148.859
C08776=1223.942,-23.095,-40.334,-179.757,5.361,148.860
C08777=1223.947,-23.345,-40.320,-179.759,5.360,148.860
C08778=1223.951,-23.595,-40.306,-179.761,5.361,148.861
C08779=1223.957,-23.844,-40.293,-179.764,5.360,148.862
C08780=1223.961,-24.094,-40.280,-179.767,5.360,148.862
C08781=1223.967,-24.343,-40.266,-179.769,5.360,148.863
C08782=1223.971,-24.593,-40.253,-179.772,5.359,148.864
C08783=1223.977,-24.843,-40.240,-179.774,5.359,148.865
C08784=1223.982,-25.092,-40.226,-179.776,5.359,148.865
C08785=1223.987,-25.342,-40.213,-179.779,5.359,148.866
C08786=1223.992,-25.591,-40.200,-179.782,5.358,148.867
C08787=1223.997,-25.841,-40.186,-179.784,5.359,148.867
C08788=1224.002,-26.091,-40.173,-179.786,5.358,148.868
C08789=1224.008,-26.340,-40.159,-179.789,5.358,148.869
C08790=1224.013,-26.589,-40.147,-179.791,5.358,148.869
C08791=1224.017,-26.839,-40.134,-179.794,5.357,148.870
C08792=1224.023,-27.088,-40.120,-179.796,5.357,148.871
C08793=1224.027,-27.339,-40.107,-179.799,5.357,148.871
C08794=1224.033,-27.588,-40.094,-179.801,5.357,148.872
C08795=1224.038,-27.838,-40.081,-179.804,5.356,148.873
C08796=1224.043,-28.087,-40.067,-179.806,5.357,148.874
C08797=1224.048,-28.337,-40.054,-179.809,5.356,148.874
C08798=1224.054,-28.587,-40.041,-179.811,5.356,148.875
C08799=1224.058,-28.836,-40.027,-179.813,5.356,148.876
C08800=1224.063,-29.086,-40.015,-179.816,5.355,148.876
C08801=1224.069,-29.335,-40.001,-179.818,5.356,148.877
C08802=1224.073,-29.585,-39.988,-179.821,5.355,148.878
C08803=1224.079,-29.834,-39.974,-179.823,5.355,148.878
C08804=1224.083,-30.084,-39.961,-179.825,5.355,148.879
C08805=1224.089,-30.334,-39.949,-179.828,5.355,148.880
C08806=1224.094,-30.584,-39.935,-179.831,5.354,148.881
C08807=1224.099,-30.833,-39.923,-179.833,5.354,148.881
C08808=1224.104,-31.082,-39.909,-179.836,5.354,148.882
C08809=1224.109,-31.332,-39.896,-179.838,5.353,148.883
C08810=1224.114,-31.582,-39.883,-179.840,5.354,148.883
C08811=1224.119,-31.832,-39.870,-179.843,5.353,148.884
C08812=1224.125,-32.081,-39.857,-179.846,5.353,148.885
C08813=1224.130,-32.330,-39.844,-179.848,5.353,148.885
C08814=1224.135,-32.580,-39.830,-179.850,5.353,148.886
C08815=1224.140,-32.829,-39.818,-179.852,5.353,148.887
C08816=1224.144,-33.080,-39.805,-179.855,5.352,148.888
C08817=1224.150,-33.329,-39.791,-179.858,5.352,148.888
C08818=1224.155,-33.578,-39.779,-179.860,5.352,148.889
C08819=1224.160,-33.828,-39.766,-179.862,5.352,148.890
C08820=1224.166,-34.078,-39.753,-179.865,5.351,148.890
C08821=1224.171,-34.327,-39.740,-179.867,5.352,148.891
C08822=1224.175,-34.577,-39.727,-179.870,5.351,148.892
C08823=1224.181,-34.826,-39.713,-179.873,5.351,148.892
C08824=1224.186,-35.076,-39.701,-179.875,5.351,148.893
C08825=1224.190,-35.326,-39.688,-179.877,5.350,148.894
C08826=1224.196,-35.575,-39.675,-179.879,5.351,148.895
C08827=1224.201,-35.825,-39.661,-179.882,5.350,148.895
C08828=1224.206,-36.075,-39.649,-179.885,5.350,148.896
C08829=1224.211,-36.324,-39.636,-179.887,5.350,148.897
C08830=1224.216,-36.574,-39.623,-179.889,5.350,148.897
C08831=1224.221,-36.824,-39.610,-179.892,5.349,148.898
C08832=1224.227,-37.073,-39.597,-179.894,5.349,148.899
C08833=1224.232,-37.322,-39.585,-179.897,5.349,148.899
C08834=1224.237,-37.573,-39.571,-179.900,5.348,148.900
C08835=1224.242,-37.822,-39.559,-179.902,5.349,148.901
C08836=1224.247,-38.071,-39.546,-179.904,5.348,148.902
C08837=1224.252,-38.321,-39.533,-179.906,5.349,148.902
C08838=1224.258,-38.571,-39.520,-179.909,5.348,148.903
C08839=1224.263,-38.820,-39.507,-179.912,5.348,148.904
C08840=1224.267,-39.070,-39.494,-179.914,5.348,148.904
C08841=1224.272,-39.320,-39.482,-179.916,5.347,148.905
C08842=1224.278,-39.569,-39.469,-179.919,5.347,148.906
C08843=1224.283,-39.819,-39.456,-179.921,5.347,148.906
C08844=1224.288,-40.069,-39.444,-179.924,5.347,148.907
C08845=1224.293,-40.319,-39.431,-179.926,5.347,148.908
C08846=1224.298,-40.568,-39.419,-179.929,5.347,148.909
C08847=1224.303,-40.818,-39.406,-179.931,5.346,148.909
C08848=1224.308,-41.067,-39.393,-179.933,5.346,148.910
C08849=1224.314,-41.317,-39.380,-179.936,5.346,148.911
C08850=1224.319,-41.566,-39.367,-179.938,5.346,148.911
C08851=1224.324,-41.816,-39.354,-179.941,5.346,148.912
C08852=1224.329,-42.065,-39.342,-179.943,5.345,148.913
C08853=1224.334,-42.315,-39.330,-179.945,5.346,148.913
C08854=1224.339,-42.565,-39.317,-179.948,5.345,148.914
C08855=1224.344,-42.815,-39.304,-179.951,5.345,148.915
C08856=1224.350,-43.064,-39.291,-179.953,5.345,148.916
C08857=1224.355,-43.314,-39.278,-179.956,5.345,148.916
C08858=1224.360,-43.563,-39.266,-179.958,5.345,148.917
C08859=1224.365,-43.814,-39.254,-179.960,5.344,148.918
C08860=1224.370,-44.063,-39.241,-179.963,5.344,148.918
C08861=1224.375,-44.312,-39.228,-179.965,5.344,148.919
C08862=1224.380,-44.562,-39.216,-179.968,5.344,148.920
C08863=1224.385,-44.812,-39.203,-179.970,5.344,148.920
C08864=1224.390,-45.062,-39.191,-179.972,5.344,148.921
C08865=1224.395,-45.311,-39.178,-179.975,5.343,148.922
C08866=1224.400,-45.560,-39.166,-179.977,5.343,148.923
C08867=1224.406,-45.810,-39.152,-179.980,5.343,148.923
C08868=1224.411,-46.060,-39.140,-179.982,5.343,148.924
C08869=1224.416,-46.310,-39.128,-179.985,5.343,148.925
C08870=1224.421,-46.559,-39.115,-179.987,5.342,148.925
C08871=1224.426,-46.808,-39.102,-179.989,5.343,148.926
C08872=1224.432,-47.058,-39.091,-179.992,5.342,148.927
C08873=1224.436,-47.308,-39.078,-179.994,5.342,148.927
C08874=1224.441,-47.558,-39.065,-179.997,5.342,148.928
C08875=1224.447,-47.807,-39.052,-179.999,5.342,148.929
C08876=1224.452,-48.057,-39.040,179.998,5.342,148.930
C08877=1224.457,-48.327,-39.027,179.996,5.341,148.930
C08878=1224.464,-48.597,-39.014,179.993,5.341,148.931
C08879=1224.469,-48.866,-39.000,179.991,5.341,148.932
C08880=1224.474,-49.136,-38.986,179.988,5.341,148.932
C08881=1224.479,-49.386,-38.974,179.986,5.340,148.933
C08882=1224.484,-49.635,-38.962,179.984,5.341,148.934
C08883=1224.489,-49.885,-38.949,179.981,5.340,148.935
C08884=1224.495,-50.135,-38.937,179.979,5.340,148.935
C08885=1224.500,-50.384,-38.925,179.976,5.340,148.936
C08886=1224.505,-50.635,-38.912,179.974,5.339,148.937
C08887=1224.510,-50.884,-38.900,179.971,5.340,148.937
C08888=1224.515,-51.133,-38.887,179.969,5.339,148.938
C08889=1224.520,-51.383,-38.875,179.967,5.340,148.939
C08890=1224.526,-51.632,-38.863,179.964,5.339,148.939
C08891=1224.531,-51.882,-38.851,179.961,5.339,148.940
C08892=1224.536,-52.132,-38.838,179.959,5.339,148.941
C08893=1224.541,-52.381,-38.826,179.957,5.339,148.942
C08894=1224.545,-52.631,-38.814,179.955,5.339,148.942
C08895=1224.550,-52.881,-38.801,179.952,5.338,148.943
C08896=1224.556,-53.131,-38.790,179.949,5.338,148.944
C08897=1224.561,-53.380,-38.777,179.947,5.338,148.944
C08898=1224.566,-53.630,-38.765,179.944,5.338,148.945
C08899=1224.572,-53.879,-38.752,179.942,5.338,148.946
C08900=1224.577,-54.129,-38.741,179.940,5.338,148.946
C08901=1224.582,-54.378,-38.728,179.938,5.338,148.947
C08902=1224.588,-54.628,-38.716,179.935,5.338,148.948
C08903=1224.592,-54.877,-38.704,179.932,5.337,148.949
C08904=1224.597,-55.128,-38.692,179.930,5.337,148.949
C08905=1224.602,-55.377,-38.679,179.927,5.337,148.950
C08906=1224.607,-55.627,-38.667,179.925,5.337,148.951
C08907=1224.612,-55.877,-38.655,179.923,5.337,148.951
C08908=1224.618,-56.127,-38.643,179.921,5.337,148.952
C08909=1224.623,-56.376,-38.630,179.918,5.337,148.953
C08910=1224.628,-56.625,-38.619,179.915,5.336,148.954
C08911=1224.633,-56.875,-38.606,179.913,5.337,148.954
C08912=1224.638,-57.125,-38.594,179.911,5.336,148.955
C08913=1224.644,-57.375,-38.583,179.908,5.336,148.956
C08914=1224.649,-57.624,-38.570,179.906,5.336,148.956
C08915=1224.654,-57.874,-38.558,179.904,5.336,148.957
C08916=1224.659,-58.123,-38.546,179.901,5.336,148.958
C08917=1224.664,-58.373,-38.534,179.898,5.335,148.958
C08918=1224.669,-58.623,-38.522,179.896,5.336,148.959
C08919=1224.675,-58.872,-38.510,179.894,5.335,148.960
C08920=1224.679,-59.122,-38.498,179.892,5.336,148.961
C08921=1224.684,-59.371,-38.486,179.889,5.335,148.961
C08922=1224.690,-59.621,-38.474,179.887,5.335,148.962
C08923=1224.695,-59.871,-38.462,179.884,5.335,148.963
C08924=1224.700,-60.120,-38.449,179.881,5.334,148.963
C08925=1224.705,-60.370,-38.438,179.879,5.335,148.964
C08926=1224.710,-60.620,-38.426,179.877,5.334,148.965
C08927=1224.715,-60.870,-38.413,179.875,5.335,148.965
C08928=1224.720,-61.120,-38.401,179.872,5.334,148.966
C08929=1224.726,-61.369,-38.390,179.870,5.335,148.967
C08930=1224.731,-61.618,-38.378,179.867,5.334,148.968
C08931=1224.736,-61.868,-38.366,179.865,5.334,148.968
C08932=1224.742,-62.118,-38.354,179.862,5.334,148.969
C08933=1224.746,-62.367,-38.343,179.860,5.333,148.970
C08934=1224.752,-62.617,-38.330,179.858,5.334,148.970
C08935=1224.757,-62.867,-38.318,179.855,5.333,148.971
C08936=1224.762,-63.116,-38.307,179.853,5.334,148.972
C08937=1224.767,-63.366,-38.295,179.850,5.333,148.973
C08938=1224.772,-63.616,-38.283,179.848,5.334,148.973
C08939=1224.777,-63.865,-38.271,179.846,5.333,148.974
C08940=1224.782,-64.115,-38.259,179.843,5.333,148.975
C08941=1224.788,-64.365,-38.247,179.841,5.333,148.975
C08942=1224.793,-64.614,-38.235,179.838,5.332,148.976
C08943=1224.798,-64.864,-38.224,179.836,5.333,148.977
C08944=1224.803,-65.114,-38.212,179.833,5.332,148.977
C08945=1224.808,-65.364,-38.200,179.831,5.333,148.978
C08946=1224.813,-65.614,-38.189,179.829,5.332,148.979
C08947=1224.818,-65.863,-38.176,179.826,5.333,148.980
C08948=1224.824,-66.113,-38.164,179.824,5.332,148.980
C08949=1224.828,-66.362,-38.153,179.821,5.332,148.981
C08950=1224.834,-66.612,-38.141,179.819,5.332,148.982
C08951=1224.839,-66.861,-38.130,179.816,5.332,148.982
C08952=1224.844,-67.111,-38.118,179.814,5.332,148.983
C08953=1224.850,-67.361,-38.105,179.812,5.331,148.984
C08954=1224.854,-67.610,-38.094,179.810,5.332,148.985
C08955=1224.860,-67.860,-38.082,179.807,5.331,148.985
C08956=1224.865,-68.110,-38.070,179.805,5.331,148.986
C08957=1224.870,-68.360,-38.059,179.803,5.331,148.986
C08958=1224.875,-68.610,-38.047,179.801,5.331,148.987
C08959=1224.880,-68.859,-38.036,179.798,5.331,148.988
C08960=1224.885,-69.109,-38.024,179.795,5.330,148.989
C08961=1224.891,-69.358,-38.013,179.793,5.331,148.989
C08962=1224.896,-69.608,-38.001,179.790,5.330,148.990
C08963=1224.901,-69.857,-37.989,179.788,5.330,148.991
C08964=1224.906,-70.107,-37.977,179.786,5.330,148.991
C08965=1224.911,-70.357,-37.965,179.784,5.330,148.992
C08966=1224.916,-70.607,-37.954,179.781,5.330,148.993
C08967=1224.922,-70.856,-37.942,179.779,5.330,148.994
C08968=1224.926,-71.106,-37.931,179.776,5.330,148.994
C08969=1224.932,-71.355,-37.919,179.774,5.330,148.995
C08970=1224.938,-71.605,-37.908,179.771,5.330,148.996
C08971=1224.942,-71.855,-37.896,179.769,5.330,148.996
C08972=1224.948,-72.105,-37.884,179.767,5.330,148.997
C08973=1224.952,-72.354,-37.873,179.764,5.329,148.998
C08974=1224.958,-72.604,-37.861,179.762,5.329,148.998
C08975=1224.963,-72.853,-37.850,179.759,5.329,148.999
C08976=1224.969,-73.103,-37.838,179.757,5.329,149.000
C08977=1224.973,-73.353,-37.827,179.754,5.329,149.001
C08978=1224.979,-73.603,-37.815,179.752,5.329,149.001
C08979=1224.983,-73.852,-37.804,179.750,5.329,149.002
C08980=1224.989,-74.102,-37.792,179.748,5.329,149.003
C08981=1224.995,-74.373,-37.780,179.745,5.329,149.003
C08982=1225.000,-74.643,-37.767,179.742,5.328,149.004
C08983=1225.006,-74.913,-37.756,179.740,5.329,149.005
C08984=1225.011,-75.184,-37.744,179.737,5.328,149.006
C08985=1225.017,-75.434,-37.732,179.735,5.329,149.007
C08986=1225.022,-75.684,-37.721,179.732,5.328,149.007
C08987=1225.028,-75.933,-37.709,179.730,5.328,149.008
C08988=1225.032,-76.182,-37.698,179.728,5.328,149.008
C08989=1225.038,-76.432,-37.686,179.725,5.327,149.009
C08990=1225.042,-76.682,-37.675,179.723,5.328,149.010
C08991=1225.048,-76.932,-37.663,179.721,5.327,149.011
C08992=1225.053,-77.181,-37.652,179.718,5.328,149.011
C08993=1225.058,-77.431,-37.641,179.716,5.327,149.012
C08994=1225.064,-77.681,-37.629,179.714,5.328,149.013
C08995=1225.068,-77.931,-37.618,179.711,5.327,149.013
C08996=1225.074,-78.180,-37.606,179.709,5.327,149.014
C08997=1225.079,-78.429,-37.595,179.706,5.327,149.015
C08998=1225.084,-78.679,-37.584,179.704,5.327,149.015
C08999=1225.089,-78.930,-37.573,179.701,5.327,149.016
C09000=1225.095,-79.179,-37.562,179.699,5.327,149.017
C09001=1225.100,-79.429,-37.550,179.697,5.327,149.018
C09002=1225.105,-79.678,-37.539,179.695,5.327,149.018
C09003=1225.110,-79.928,-37.527,179.692,5.327,149.019
C09004=1225.116,-80.178,-37.517,179.690,5.327,149.020
C09005=1225.121,-80.427,-37.505,179.687,5.327,149.020
C09006=1225.125,-80.677,-37.494,179.685,5.327,149.021
C09007=1225.131,-80.927,-37.482,179.682,5.326,149.022
C09008=1225.136,-81.176,-37.472,179.680,5.327,149.023
C09009=1225.141,-81.426,-37.461,179.678,5.326,149.023
C09010=1225.146,-81.676,-37.449,179.675,5.326,149.024
C09011=1225.152,-81.925,-37.438,179.673,5.326,149.024
C09012=1225.157,-82.175,-37.427,179.671,5.325,149.025
C09013=1225.162,-82.425,-37.415,179.669,5.326,149.026
C09014=1225.167,-82.675,-37.404,179.666,5.325,149.027
C09015=1225.172,-82.924,-37.394,179.664,5.326,149.027
C09016=1225.178,-83.174,-37.382,179.661,5.325,149.028
C09017=1225.183,-83.424,-37.371,179.659,5.326,149.029
C09018=1225.188,-83.673,-37.360,179.656,5.325,149.029
C09019=1225.193,-83.923,-37.349,179.654,5.326,149.030
C09020=1225.198,-84.173,-37.337,179.652,5.325,149.031
C09021=1225.204,-84.422,-37.326,179.650,5.325,149.032
C09022=1225.209,-84.672,-37.316,179.647,5.325,149.032
C09023=1225.214,-84.922,-37.304,179.645,5.325,149.033
C09024=1225.219,-85.172,-37.293,179.642,5.325,149.034
C09025=1225.224,-85.421,-37.282,179.640,5.325,149.034
C09026=1225.229,-85.671,-37.271,179.637,5.325,149.035
C09027=1225.235,-85.921,-37.260,179.635,5.325,149.036
C09028=1225.240,-86.170,-37.249,179.633,5.325,149.037
C09029=1225.245,-86.420,-37.238,179.631,5.325,149.037
C09030=1225.250,-86.669,-37.227,179.628,5.324,149.038
C09031=1225.256,-86.919,-37.216,179.626,5.325,149.038
C09032=1225.261,-87.170,-37.205,179.624,5.324,149.039
C09033=1225.266,-87.418,-37.194,179.622,5.324,149.040
C09034=1225.271,-87.668,-37.183,179.619,5.324,149.041
C09035=1225.276,-87.918,-37.172,179.617,5.324,149.041
C09036=1225.282,-88.168,-37.161,179.614,5.324,149.042
C09037=1225.287,-88.418,-37.150,179.612,5.324,149.043
C09038=1225.291,-88.667,-37.139,179.609,5.324,149.043
C09039=1225.297,-88.917,-37.129,179.607,5.324,149.044
C09040=1225.302,-89.167,-37.117,179.605,5.324,149.045
C09041=1225.308,-89.417,-37.107,179.602,5.324,149.046
C09042=1225.313,-89.666,-37.095,179.600,5.324,149.046
C09043=1225.318,-89.916,-37.085,179.598,5.324,149.047
C09044=1225.323,-90.165,-37.074,179.595,5.324,149.048
C09045=1225.328,-90.416,-37.063,179.593,5.324,149.048
C09046=1225.333,-90.664,-37.052,179.591,5.323,149.049
C09047=1225.338,-90.915,-37.042,179.589,5.323,149.050
C09048=1225.344,-91.165,-37.030,179.586,5.323,149.050
C09049=1225.349,-91.414,-37.020,179.584,5.323,149.051
C09050=1225.354,-91.664,-37.008,179.581,5.323,149.052
C09051=1225.360,-91.913,-36.998,179.579,5.323,149.052
C09052=1225.364,-92.163,-36.987,179.576,5.323,149.053
C09053=1225.369,-92.413,-36.976,179.574,5.323,149.054
C09054=1225.375,-92.662,-36.965,179.572,5.323,149.055
C09055=1225.380,-92.913,-36.954,179.570,5.323,149.055
C09056=1225.386,-93.162,-36.944,179.567,5.323,149.056
C09057=1225.391,-93.412,-36.933,179.565,5.323,149.057
C09058=1225.396,-93.661,-36.922,179.562,5.323,149.057
C09059=1225.401,-93.911,-36.911,179.560,5.323,149.058
C09060=1225.406,-94.161,-36.901,179.558,5.322,149.059
C09061=1225.412,-94.411,-36.890,179.556,5.323,149.059
C09062=1225.416,-94.660,-36.879,179.553,5.322,149.060
C09063=1225.422,-94.910,-36.869,179.551,5.322,149.061
C09064=1225.427,-95.160,-36.858,179.548,5.322,149.061
C09065=1225.432,-95.409,-36.847,179.546,5.322,149.062
C09066=1225.437,-95.659,-36.837,179.544,5.322,149.063
C09067=1225.443,-95.909,-36.825,179.541,5.322,149.064
C09068=1225.448,-96.159,-36.815,179.539,5.322,149.064
C09069=1225.454,-96.408,-36.804,179.537,5.322,149.065
C09070=1225.458,-96.658,-36.793,179.534,5.322,149.066
C09071=1225.464,-96.908,-36.783,179.532,5.322,149.066
C09072=1225.469,-97.158,-36.772,179.530,5.321,149.067
C09073=1225.475,-97.407,-36.762,179.528,5.322,149.068
C09074=1225.479,-97.657,-36.751,179.525,5.321,149.068
C09075=1225.485,-97.907,-36.741,179.523,5.322,149.069
C09076=1225.490,-98.157,-36.730,179.520,5.321,149.070
C09077=1225.495,-98.406,-36.719,179.518,5.322,149.071
C09078=1225.500,-98.656,-36.709,179.516,5.322,149.071
C09079=1225.506,-98.906,-36.698,179.513,5.321,149.072
C09080=1225.511,-99.156,-36.688,179.511,5.322,149.073
C09081=1225.516,-99.405,-36.677,179.509,5.321,149.073
C09082=1225.521,-99.655,-36.666,179.507,5.322,149.074
C09083=1225.527,-99.904,-36.656,179.504,5.321,149.075
C09084=1225.532,-100.155,-36.646,179.502,5.321,149.075
C09085=1225.537,-100.425,-36.634,179.499,5.321,149.076
C09086=1225.543,-100.696,-36.623,179.496,5.321,149.077
C09087=1225.548,-100.968,-36.612,179.494,5.321,149.078
C09088=1225.554,-101.239,-36.600,179.492,5.321,149.078
C09089=1225.559,-101.488,-36.589,179.490,5.321,149.079
C09090=1225.565,-101.738,-36.579,179.487,5.321,149.080
C09091=1225.570,-101.988,-36.569,179.485,5.321,149.080
C09092=1225.576,-102.237,-36.558,179.482,5.321,149.081
C09093=1225.580,-102.487,-36.548,179.480,5.321,149.082
C09094=1225.585,-102.736,-36.537,179.478,5.320,149.082
C09095=1225.590,-102.987,-36.527,179.476,5.321,149.083
C09096=1225.596,-103.236,-36.517,179.473,5.320,149.084
C09097=1225.601,-103.486,-36.506,179.471,5.320,149.085
C09098=1225.606,-103.736,-36.496,179.468,5.320,149.085
C09099=1225.612,-103.985,-36.485,179.466,5.320,149.086
C09100=1225.617,-104.235,-36.474,179.464,5.320,149.087
C09101=1225.622,-104.485,-36.464,179.461,5.320,149.087
C09102=1225.627,-104.735,-36.454,179.459,5.321,149.088
C09103=1225.632,-104.984,-36.444,179.457,5.320,149.089
C09104=1225.638,-105.234,-36.434,179.455,5.320,149.089
C09105=1225.643,-105.484,-36.423,179.452,5.320,149.090
C09106=1225.648,-105.733,-36.413,179.450,5.320,149.091
C09107=1225.653,-105.984,-36.402,179.448,5.320,149.091
C09108=1225.659,-106.233,-36.392,179.446,5.320,149.092
C09109=1225.664,-106.482,-36.383,179.443,5.320,149.093
C09110=1225.669,-106.733,-36.372,179.441,5.320,149.094
C09111=1225.674,-106.982,-36.361,179.438,5.320,149.094
C09112=1225.679,-107.232,-36.350,179.436,5.320,149.095
C09113=1225.685,-107.481,-36.340,179.434,5.319,149.096
C09114=1225.690,-107.731,-36.330,179.432,5.320,149.096
C09115=1225.695,-107.981,-36.320,179.429,5.319,149.097
C09116=1225.700,-108.230,-36.310,179.427,5.320,149.098
C09117=1225.706,-108.480,-36.300,179.424,5.319,149.098
C09118=1225.711,-108.730,-36.289,179.422,5.319,149.099
C09119=1225.716,-108.980,-36.279,179.420,5.320,149.100
C09120=1225.721,-109.230,-36.269,179.418,5.319,149.100
C09121=1225.726,-109.479,-36.259,179.416,5.319,149.101
C09122=1225.732,-109.729,-36.249,179.413,5.319,149.102
C09123=1225.737,-109.979,-36.238,179.411,5.319,149.102
C09124=1225.743,-110.229,-36.228,179.408,5.319,149.103
C09125=1225.748,-110.478,-36.219,179.406,5.319,149.104
C09126=1225.753,-110.729,-36.208,179.404,5.319,149.105
C09127=1225.758,-110.978,-36.198,179.401,5.319,149.105
C09128=1225.764,-111.228,-36.188,179.399,5.318,149.106
C09129=1225.768,-111.478,-36.178,179.397,5.319,149.106
C09130=1225.774,-111.727,-36.168,179.395,5.318,149.107
C09131=1225.779,-111.977,-36.157,179.392,5.319,149.108
C09132=1225.784,-112.227,-36.147,179.390,5.318,149.109
C09133=1225.789,-112.476,-36.137,179.388,5.319,149.109
